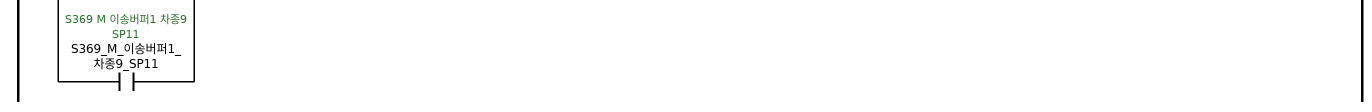
(* [picture p288: S369_유틸리티 rungs L95-L95] *)
(* S369_이송버퍼01 차종 유 *)
(* Rung L95 *)
IF (S369_M_이송버퍼1_차종1_AX OR S369_M_이송버퍼1_차종1_B OR S369_M_이송버퍼1_차종1_C OR S369_M_이송버퍼1_차종1_D OR S369_M_이송버퍼1_차종1_E OR S369_M_이송버퍼1_차종1_F OR S369_M_이송버퍼1_차종1_G OR S369_M_이송버퍼1_차종1_H) AND (S369_M_이송버퍼1_차종2_3DR OR S369_M_이송버퍼1_차종2_4DR OR S369_M_이송버퍼1_차종2_5DR OR S369_M_이송버퍼1_차종2_WGN OR S369_M_이송버퍼1_차종2_SP1 OR S369_M_이송버퍼1_차종2_SP2) AND (S369_M_이송버퍼1_차종3_LHD OR S369_M_이송버퍼1_차종3_RHD) AND (S369_M_이송버퍼1_차종4_내수 OR S369_M_이송버퍼1_차종4_수출 OR S369_M_이송버퍼1_차종4_북미 OR S369_M_이송버퍼1_차종4_EEC OR S369_M_이송버퍼1_차종4_호주 OR S369_M_이송버퍼1_차종4_중동 OR S369_M_이송버퍼1_차종4_중국 OR S369_M_이송버퍼1_차종4_브라질 OR S369_M_이송버퍼1_차종4_SP1 OR S369_M_이송버퍼1_차종4_SP2 OR S369_M_이송버퍼1_차종4_러시아 OR S369_M_이송버퍼1_차종4_SP3 OR S369_M_이송버퍼1_차종4_SP4 OR S369_M_이송버퍼1_차종4_SP5 OR S369_M_이송버퍼1_차종4_SP6 OR S369_M_이송버퍼1_차종4_SP7) AND (S369_M_이송버퍼1_차종5_MT OR S369_M_이송버퍼1_차종5_AT OR S369_M_이송버퍼1_차종5_SP1) AND (S369_M_이송버퍼1_차종6_일반루프 OR S369_M_이송버퍼1_차종6_썬루프 OR S369_M_이송버퍼1_차종6_파노라마루프 OR S369_M_이송버퍼1_차종6_DSROOF OR S369_M_이송버퍼1_차종6_SP1) AND (S369_M_이송버퍼1_차종7_GSL OR S369_M_이송버퍼1_차종7_DSL OR S369_M_이송버퍼1_차종7_SP1 OR S369_M_이송버퍼1_차종7_SP2 OR S369_M_이송버퍼1_차종7_SP3 OR S369_M_이송버퍼1_차종7_SP4 OR S369_M_이송버퍼1_차종7_SP5 OR S369_M_이송버퍼1_차종7_SP6) AND (S369_M_이송버퍼1_차종8_2WD OR S369_M_이송버퍼1_차종8_4WD OR S369_M_이송버퍼1_차종8_SP1) AND (S369_M_이송버퍼1_차종9_MPI OR S369_M_이송버퍼1_차종9_T_GDI OR S369_M_이송버퍼1_차종9_SP1 OR S369_M_이송버퍼1_차종9_SP2 OR S369_M_이송버퍼1_차종9_SP3 OR S369_M_이송버퍼1_차종9_SP4 OR S369_M_이송버퍼1_차종9_SP5 OR S369_M_이송버퍼1_차종9_SP6 OR S369_M_이송버퍼1_차종9_SP7 OR S369_M_이송버퍼1_차종9_SP8 OR S369_M_이송버퍼1_차종9_SP9 OR S369_M_이송버퍼1_차종9_SP10 OR S369_M_이송버퍼1_차종9_SP11) AND (S369_M_이송버퍼1_차종_OPT1_슬라이딩_유 OR S369_M_이송버퍼1_차종_OPT1_슬라이딩_무 OR S369_M_이송버퍼1_차종_OPT1_R_RACK_유 OR S369_M_이송버퍼1_차종_OPT1_R_RACK_무 OR S369_M_이송버퍼1_차종_OPT1_폴딩_유 OR S369_M_이송버퍼1_차종_OPT1_폴딩_무 OR S369_M_이송버퍼1_차종_OPT1_S_REP_EATER_유 OR S369_M_이송버퍼1_차종_OPT1_S_REP_EATER_무 OR S369_M_이송버퍼1_차종_OPT1_VAN_유 OR S369_M_이송버퍼1_차종_OPT1_VAN_무) THEN
    _t5 := S369_M_이송버퍼1_SEQ <> 0;
END_IF;
S369_M_이송버퍼1_차종_유 := _t5;

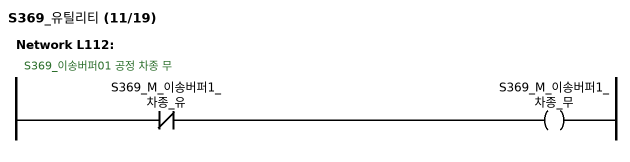
(* S369_이송버퍼01 공정 차종 무 *)
(* Rung L112 *)
S369_M_이송버퍼1_차종_무 := NOT S369_M_이송버퍼1_차종_유;

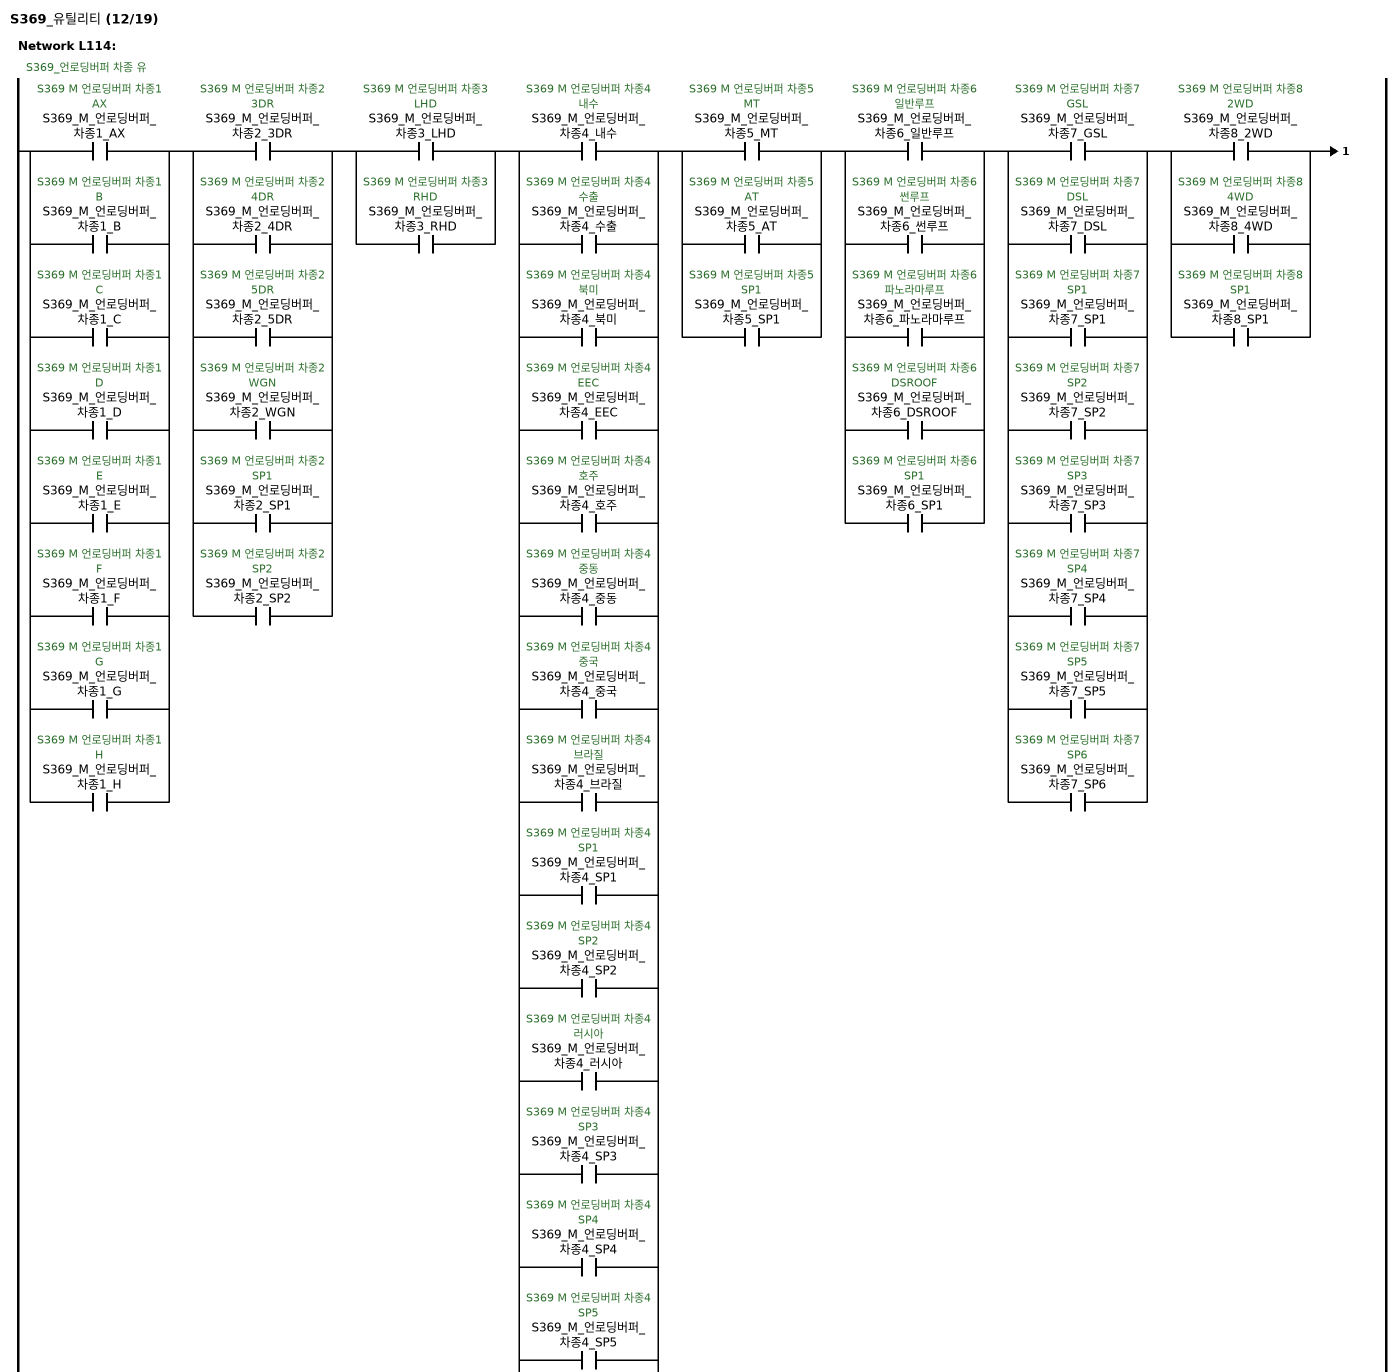

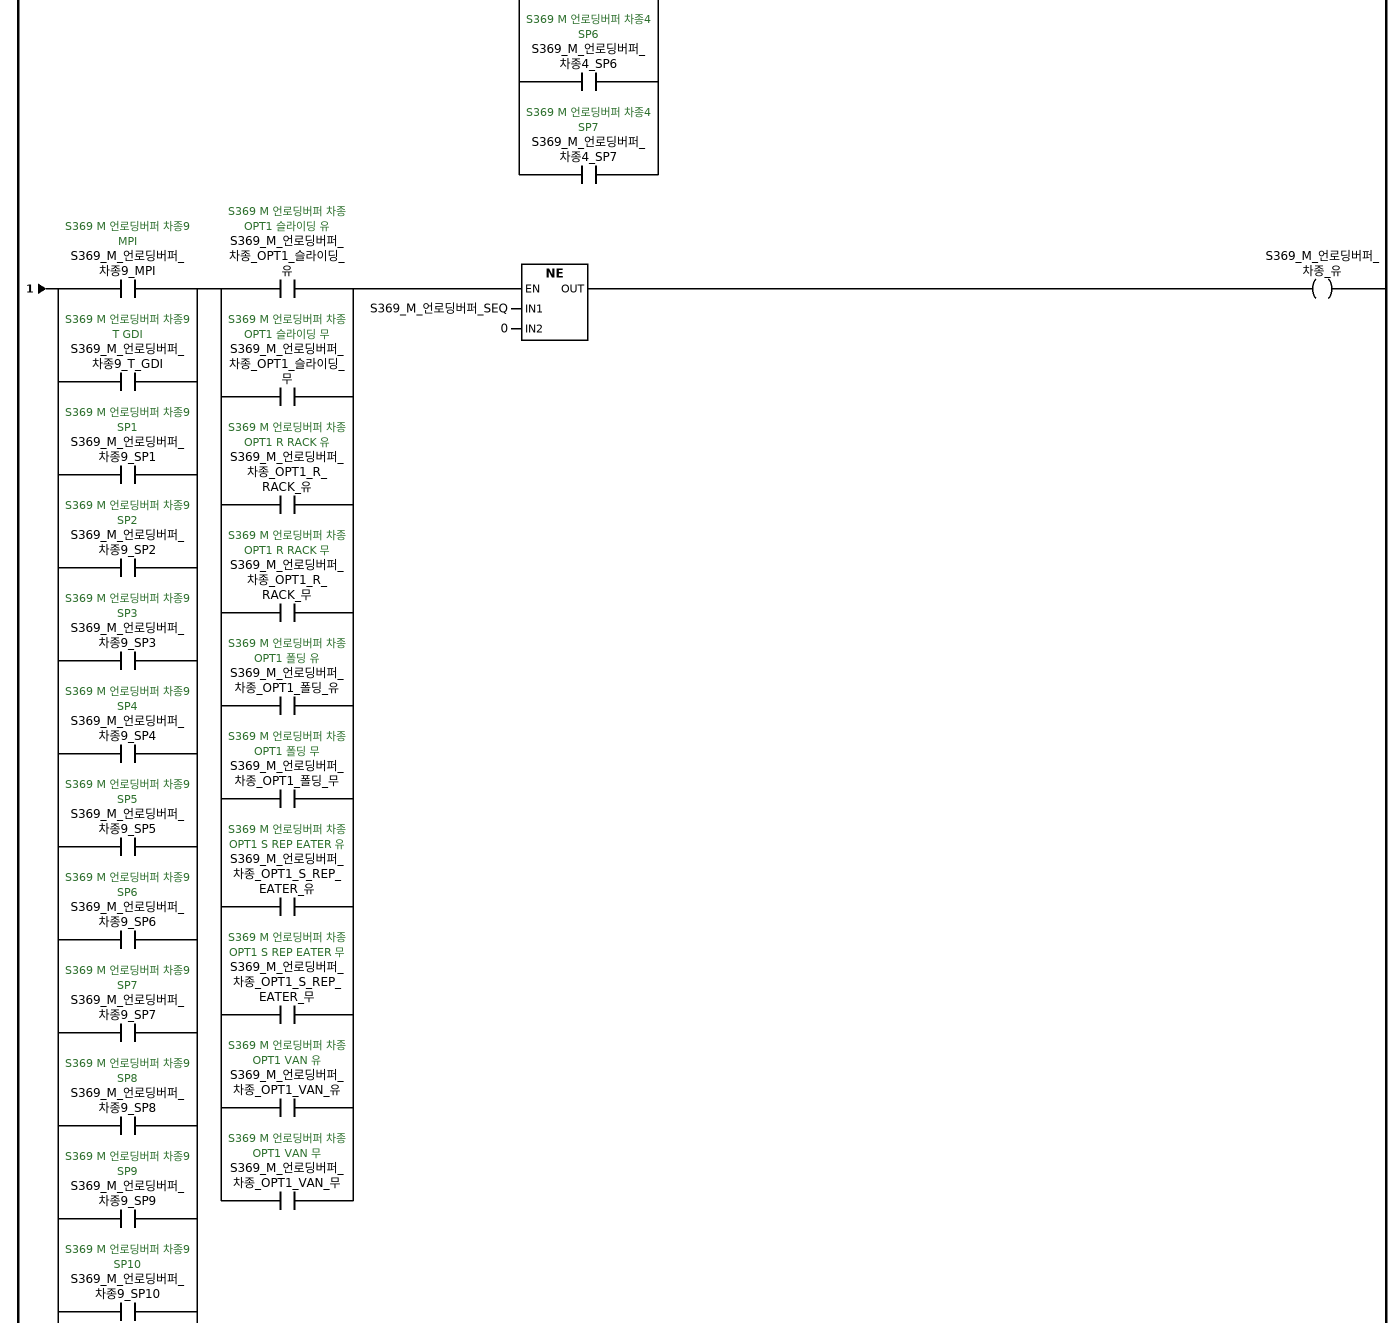

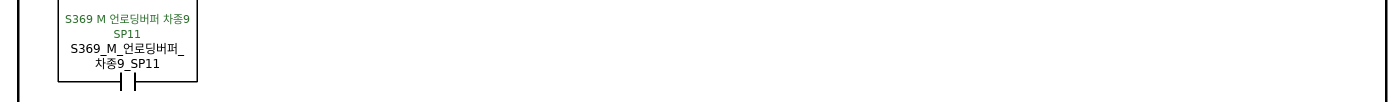
(* S369_언로딩버퍼 차종 유 *)
(* Rung L114 *)
IF (S369_M_언로딩버퍼_차종1_AX OR S369_M_언로딩버퍼_차종1_B OR S369_M_언로딩버퍼_차종1_C OR S369_M_언로딩버퍼_차종1_D OR S369_M_언로딩버퍼_차종1_E OR S369_M_언로딩버퍼_차종1_F OR S369_M_언로딩버퍼_차종1_G OR S369_M_언로딩버퍼_차종1_H) AND (S369_M_언로딩버퍼_차종2_3DR OR S369_M_언로딩버퍼_차종2_4DR OR S369_M_언로딩버퍼_차종2_5DR OR S369_M_언로딩버퍼_차종2_WGN OR S369_M_언로딩버퍼_차종2_SP1 OR S369_M_언로딩버퍼_차종2_SP2) AND (S369_M_언로딩버퍼_차종3_LHD OR S369_M_언로딩버퍼_차종3_RHD) AND (S369_M_언로딩버퍼_차종4_내수 OR S369_M_언로딩버퍼_차종4_수출 OR S369_M_언로딩버퍼_차종4_북미 OR S369_M_언로딩버퍼_차종4_EEC OR S369_M_언로딩버퍼_차종4_호주 OR S369_M_언로딩버퍼_차종4_중동 OR S369_M_언로딩버퍼_차종4_중국 OR S369_M_언로딩버퍼_차종4_브라질 OR S369_M_언로딩버퍼_차종4_SP1 OR S369_M_언로딩버퍼_차종4_SP2 OR S369_M_언로딩버퍼_차종4_러시아 OR S369_M_언로딩버퍼_차종4_SP3 OR S369_M_언로딩버퍼_차종4_SP4 OR S369_M_언로딩버퍼_차종4_SP5 OR S369_M_언로딩버퍼_차종4_SP6 OR S369_M_언로딩버퍼_차종4_SP7) AND (S369_M_언로딩버퍼_차종5_MT OR S369_M_언로딩버퍼_차종5_AT OR S369_M_언로딩버퍼_차종5_SP1) AND (S369_M_언로딩버퍼_차종6_일반루프 OR S369_M_언로딩버퍼_차종6_썬루프 OR S369_M_언로딩버퍼_차종6_파노라마루프 OR S369_M_언로딩버퍼_차종6_DSROOF OR S369_M_언로딩버퍼_차종6_SP1) AND (S369_M_언로딩버퍼_차종7_GSL OR S369_M_언로딩버퍼_차종7_DSL OR S369_M_언로딩버퍼_차종7_SP1 OR S369_M_언로딩버퍼_차종7_SP2 OR S369_M_언로딩버퍼_차종7_SP3 OR S369_M_언로딩버퍼_차종7_SP4 OR S369_M_언로딩버퍼_차종7_SP5 OR S369_M_언로딩버퍼_차종7_SP6) AND (S369_M_언로딩버퍼_차종8_2WD OR S369_M_언로딩버퍼_차종8_4WD OR S369_M_언로딩버퍼_차종8_SP1) AND (S369_M_언로딩버퍼_차종9_MPI OR S369_M_언로딩버퍼_차종9_T_GDI OR S369_M_언로딩버퍼_차종9_SP1 OR S369_M_언로딩버퍼_차종9_SP2 OR S369_M_언로딩버퍼_차종9_SP3 OR S369_M_언로딩버퍼_차종9_SP4 OR S369_M_언로딩버퍼_차종9_SP5 OR S369_M_언로딩버퍼_차종9_SP6 OR S369_M_언로딩버퍼_차종9_SP7 OR S369_M_언로딩버퍼_차종9_SP8 OR S369_M_언로딩버퍼_차종9_SP9 OR S369_M_언로딩버퍼_차종9_SP10 OR S369_M_언로딩버퍼_차종9_SP11) AND (S369_M_언로딩버퍼_차종_OPT1_슬라이딩_유 OR S369_M_언로딩버퍼_차종_OPT1_슬라이딩_무 OR S369_M_언로딩버퍼_차종_OPT1_R_RACK_유 OR S369_M_언로딩버퍼_차종_OPT1_R_RACK_무 OR S369_M_언로딩버퍼_차종_OPT1_폴딩_유 OR S369_M_언로딩버퍼_차종_OPT1_폴딩_무 OR S369_M_언로딩버퍼_차종_OPT1_S_REP_EATER_유 OR S369_M_언로딩버퍼_차종_OPT1_S_REP_EATER_무 OR S369_M_언로딩버퍼_차종_OPT1_VAN_유 OR S369_M_언로딩버퍼_차종_OPT1_VAN_무) THEN
    _t6 := S369_M_언로딩버퍼_SEQ <> 0;
END_IF;
S369_M_언로딩버퍼_차종_유 := _t6;

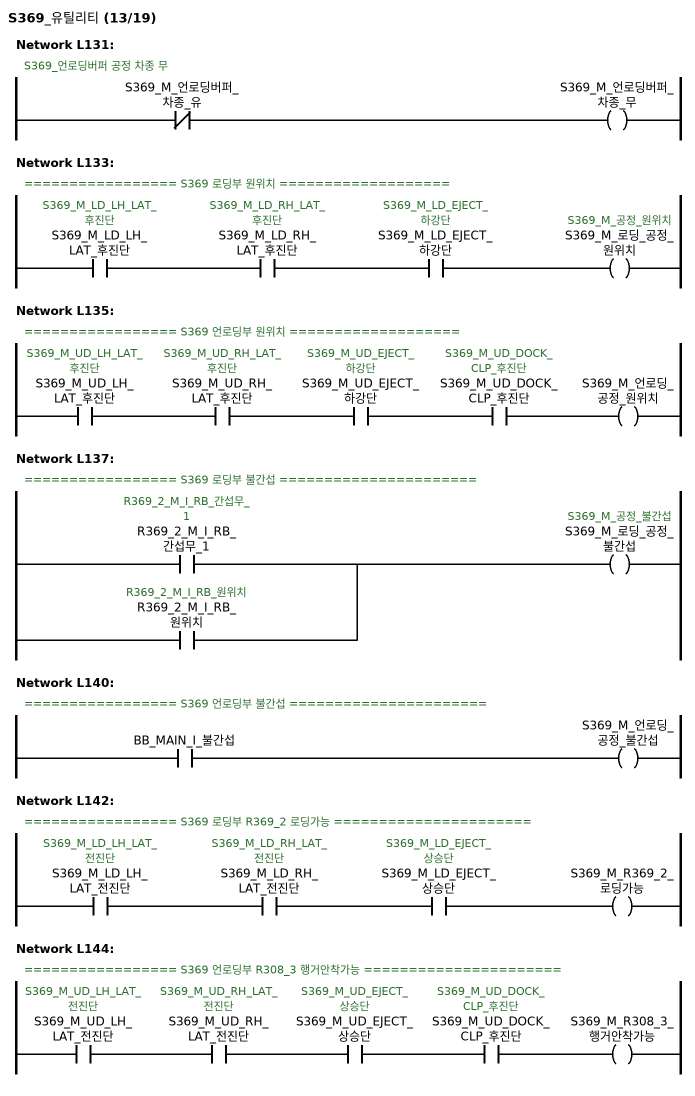
(* S369_언로딩버퍼 공정 차종 무 *)
(* Rung L131 *)
S369_M_언로딩버퍼_차종_무 := NOT S369_M_언로딩버퍼_차종_유;
(* ================= S369 로딩부 원위치 =================== *)
(* Rung L133 *)
S369_M_로딩_공정_원위치 := S369_M_LD_LH_LAT_후진단 AND S369_M_LD_RH_LAT_후진단 AND S369_M_LD_EJECT_하강단;
(* ================= S369 언로딩부 원위치 =================== *)
(* Rung L135 *)
S369_M_언로딩_공정_원위치 := S369_M_UD_LH_LAT_후진단 AND S369_M_UD_RH_LAT_후진단 AND S369_M_UD_EJECT_하강단 AND S369_M_UD_DOCK_CLP_후진단;
(* ================= S369 로딩부 불간섭 ====================== *)
(* Rung L137 *)
S369_M_로딩_공정_불간섭 := R369_2_M_I_RB_간섭무_1 OR R369_2_M_I_RB_원위치;
(* ================= S369 언로딩부 불간섭 ====================== *)
(* Rung L140 *)
S369_M_언로딩_공정_불간섭 := BB_MAIN_I_불간섭;
(* ================= S369 로딩부 R369_2 로딩가능 ====================== *)
(* Rung L142 *)
S369_M_R369_2_로딩가능 := S369_M_LD_LH_LAT_전진단 AND S369_M_LD_RH_LAT_전진단 AND S369_M_LD_EJECT_상승단;
(* ================= S369 언로딩부 R308_3 행거안착가능 ====================== *)
(* Rung L144 *)
S369_M_R308_3_행거안착가능 := S369_M_UD_LH_LAT_전진단 AND S369_M_UD_RH_LAT_전진단 AND S369_M_UD_EJECT_상승단 AND S369_M_UD_DOCK_CLP_후진단;

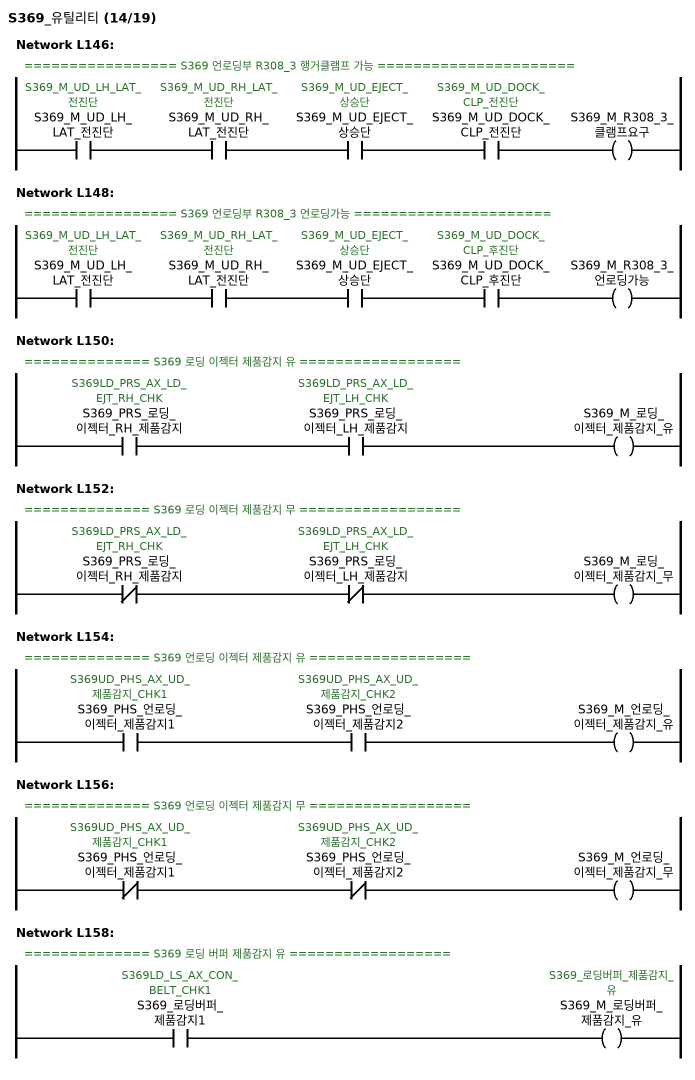
(* ================= S369 언로딩부 R308_3 행거클램프 가능 ====================== *)
(* Rung L146 *)
S369_M_R308_3_클램프요구 := S369_M_UD_LH_LAT_전진단 AND S369_M_UD_RH_LAT_전진단 AND S369_M_UD_EJECT_상승단 AND S369_M_UD_DOCK_CLP_전진단;
(* ================= S369 언로딩부 R308_3 언로딩가능 ====================== *)
(* Rung L148 *)
S369_M_R308_3_언로딩가능 := S369_M_UD_LH_LAT_전진단 AND S369_M_UD_RH_LAT_전진단 AND S369_M_UD_EJECT_상승단 AND S369_M_UD_DOCK_CLP_후진단;
(* ============== S369 로딩 이젝터 제품감지 유 ================== *)
(* Rung L150 *)
S369_M_로딩_이젝터_제품감지_유 := S369_PRS_로딩_이젝터_RH_제품감지 AND S369_PRS_로딩_이젝터_LH_제품감지;
(* ============== S369 로딩 이젝터 제품감지 무 ================== *)
(* Rung L152 *)
S369_M_로딩_이젝터_제품감지_무 := NOT S369_PRS_로딩_이젝터_RH_제품감지 AND NOT S369_PRS_로딩_이젝터_LH_제품감지;
(* ============== S369 언로딩 이젝터 제품감지 유 ================== *)
(* Rung L154 *)
S369_M_언로딩_이젝터_제품감지_유 := S369_PHS_언로딩_이젝터_제품감지1 AND S369_PHS_언로딩_이젝터_제품감지2;
(* ============== S369 언로딩 이젝터 제품감지 무 ================== *)
(* Rung L156 *)
S369_M_언로딩_이젝터_제품감지_무 := NOT S369_PHS_언로딩_이젝터_제품감지1 AND NOT S369_PHS_언로딩_이젝터_제품감지2;
(* ============== S369 로딩 버퍼 제품감지 유 ================== *)
(* Rung L158 *)
S369_M_로딩버퍼_제품감지_유 := S369_로딩버퍼_제품감지1;

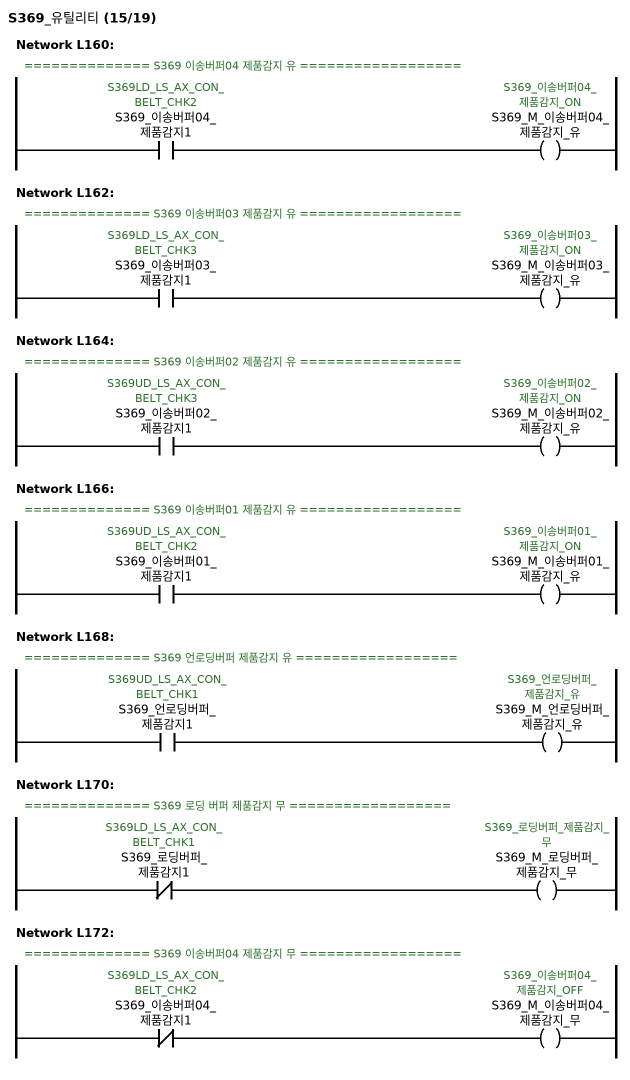
(* ============== S369 이송버퍼04 제품감지 유 ================== *)
(* Rung L160 *)
S369_M_이송버퍼04_제품감지_유 := S369_이송버퍼04_제품감지1;
(* ============== S369 이송버퍼03 제품감지 유 ================== *)
(* Rung L162 *)
S369_M_이송버퍼03_제품감지_유 := S369_이송버퍼03_제품감지1;
(* ============== S369 이송버퍼02 제품감지 유 ================== *)
(* Rung L164 *)
S369_M_이송버퍼02_제품감지_유 := S369_이송버퍼02_제품감지1;
(* ============== S369 이송버퍼01 제품감지 유 ================== *)
(* Rung L166 *)
S369_M_이송버퍼01_제품감지_유 := S369_이송버퍼01_제품감지1;
(* ============== S369 언로딩버퍼 제품감지 유 ================== *)
(* Rung L168 *)
S369_M_언로딩버퍼_제품감지_유 := S369_언로딩버퍼_제품감지1;
(* ============== S369 로딩 버퍼 제품감지 무 ================== *)
(* Rung L170 *)
S369_M_로딩버퍼_제품감지_무 := NOT S369_로딩버퍼_제품감지1;
(* ============== S369 이송버퍼04 제품감지 무 ================== *)
(* Rung L172 *)
S369_M_이송버퍼04_제품감지_무 := NOT S369_이송버퍼04_제품감지1;

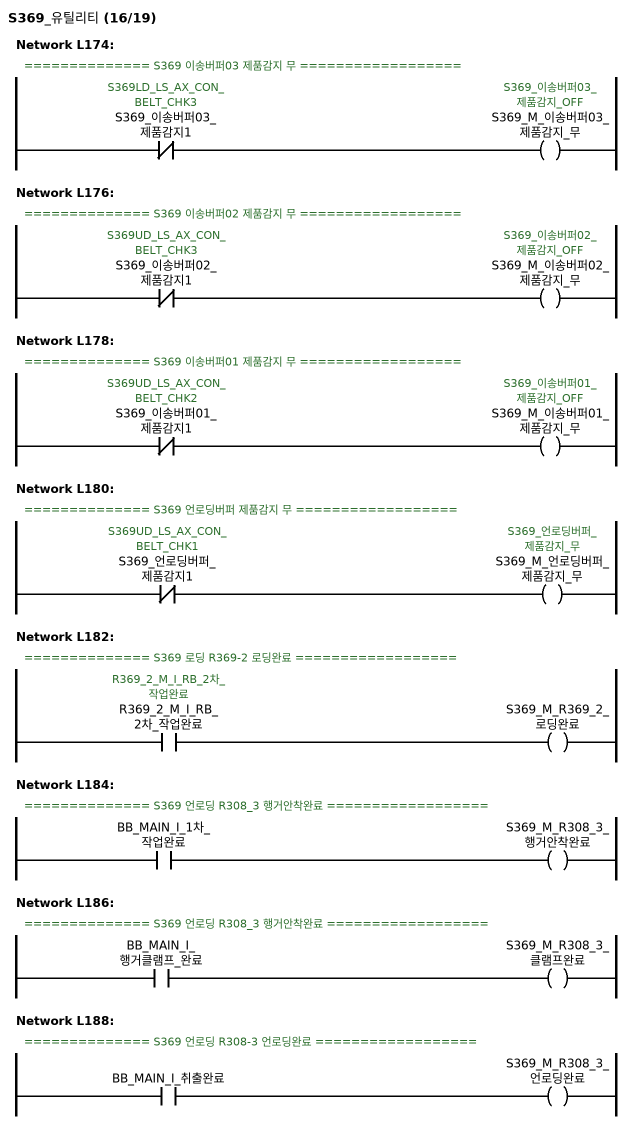
(* ============== S369 이송버퍼03 제품감지 무 ================== *)
(* Rung L174 *)
S369_M_이송버퍼03_제품감지_무 := NOT S369_이송버퍼03_제품감지1;
(* ============== S369 이송버퍼02 제품감지 무 ================== *)
(* Rung L176 *)
S369_M_이송버퍼02_제품감지_무 := NOT S369_이송버퍼02_제품감지1;
(* ============== S369 이송버퍼01 제품감지 무 ================== *)
(* Rung L178 *)
S369_M_이송버퍼01_제품감지_무 := NOT S369_이송버퍼01_제품감지1;
(* ============== S369 언로딩버퍼 제품감지 무 ================== *)
(* Rung L180 *)
S369_M_언로딩버퍼_제품감지_무 := NOT S369_언로딩버퍼_제품감지1;
(* ============== S369 로딩 R369-2 로딩완료 ================== *)
(* Rung L182 *)
S369_M_R369_2_로딩완료 := R369_2_M_I_RB_2차_작업완료;
(* ============== S369 언로딩 R308_3 행거안착완료 ================== *)
(* Rung L184 *)
S369_M_R308_3_행거안착완료 := BB_MAIN_I_1차_작업완료;
(* ============== S369 언로딩 R308_3 행거안착완료 ================== *)
(* Rung L186 *)
S369_M_R308_3_클램프완료 := BB_MAIN_I_행거클램프_완료;
(* ============== S369 언로딩 R308-3 언로딩완료 ================== *)
(* Rung L188 *)
S369_M_R308_3_언로딩완료 := BB_MAIN_I_취출완료;

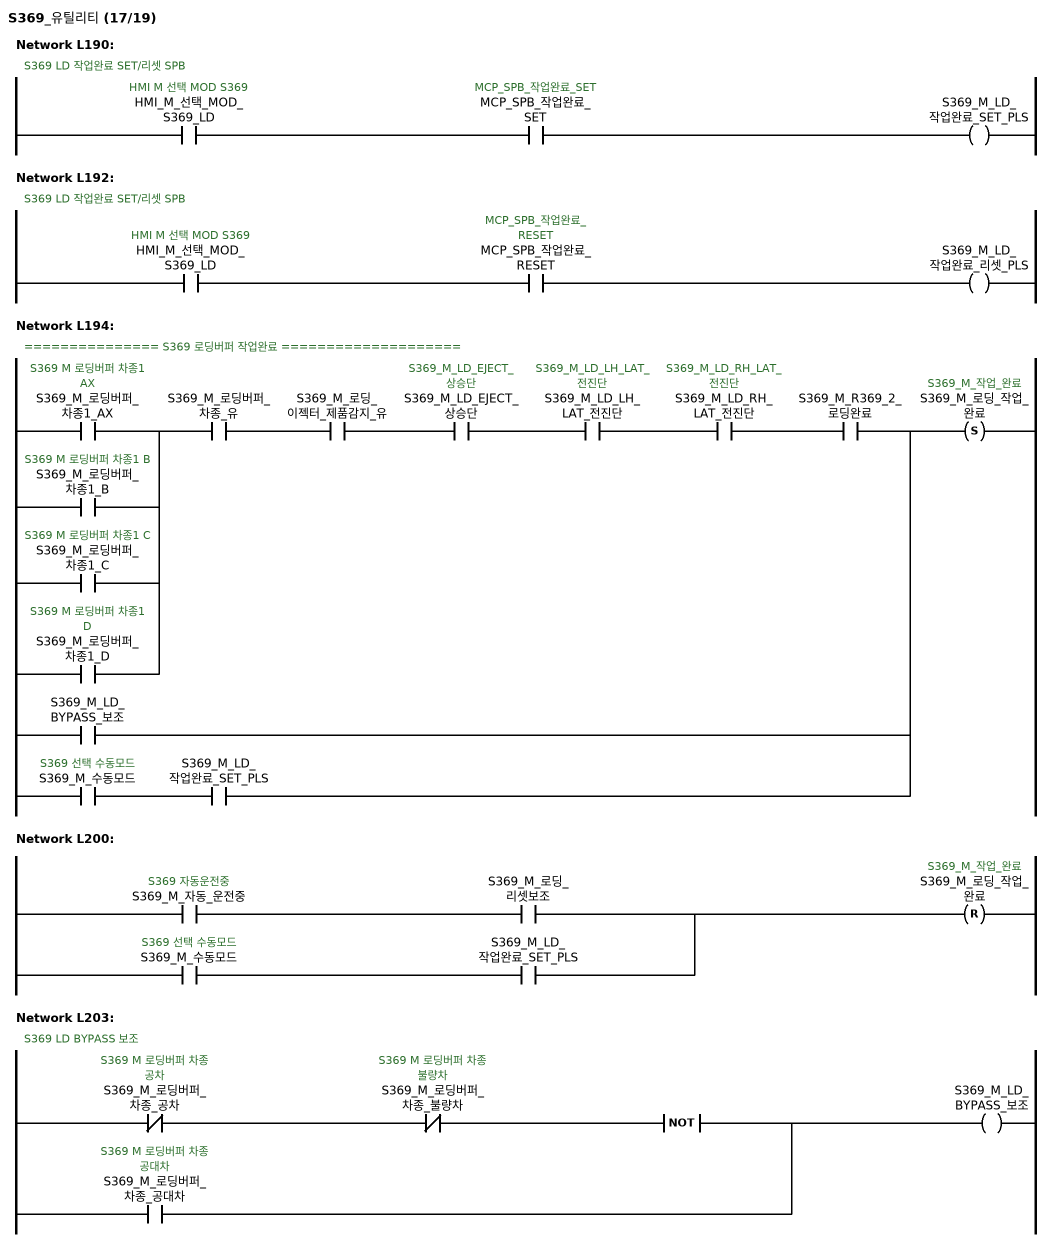
(* S369 LD 작업완료 SET/리셋 SPB *)
(* Rung L190 *)
S369_M_LD_작업완료_SET_PLS := HMI_M_선택_MOD_S369_LD AND MCP_SPB_작업완료_SET;
(* S369 LD 작업완료 SET/리셋 SPB *)
(* Rung L192 *)
S369_M_LD_작업완료_리셋_PLS := HMI_M_선택_MOD_S369_LD AND MCP_SPB_작업완료_RESET;
(* =============== S369 로딩버퍼 작업완료 ==================== *)
(* Rung L194 *)
IF ((S369_M_로딩버퍼_차종1_AX OR S369_M_로딩버퍼_차종1_B OR S369_M_로딩버퍼_차종1_C OR S369_M_로딩버퍼_차종1_D) AND S369_M_로딩버퍼_차종_유 AND S369_M_로딩_이젝터_제품감지_유 AND S369_M_LD_EJECT_상승단 AND S369_M_LD_LH_LAT_전진단 AND S369_M_LD_RH_LAT_전진단 AND S369_M_R369_2_로딩완료) OR S369_M_LD_BYPASS_보조 OR (S369_M_수동모드 AND S369_M_LD_작업완료_SET_PLS) THEN
    S369_M_로딩_작업_완료 := TRUE;
END_IF;
(* Rung L200 *)
IF (S369_M_자동_운전중 AND S369_M_로딩_리셋보조) OR (S369_M_수동모드 AND S369_M_LD_작업완료_SET_PLS) THEN
    S369_M_로딩_작업_완료 := FALSE;
END_IF;
(* S369 LD BYPASS 보조 *)
(* Rung L203 *)
S369_M_LD_BYPASS_보조 := NOT (NOT S369_M_로딩버퍼_차종_공차 AND NOT S369_M_로딩버퍼_차종_불량차) OR S369_M_로딩버퍼_차종_공대차;

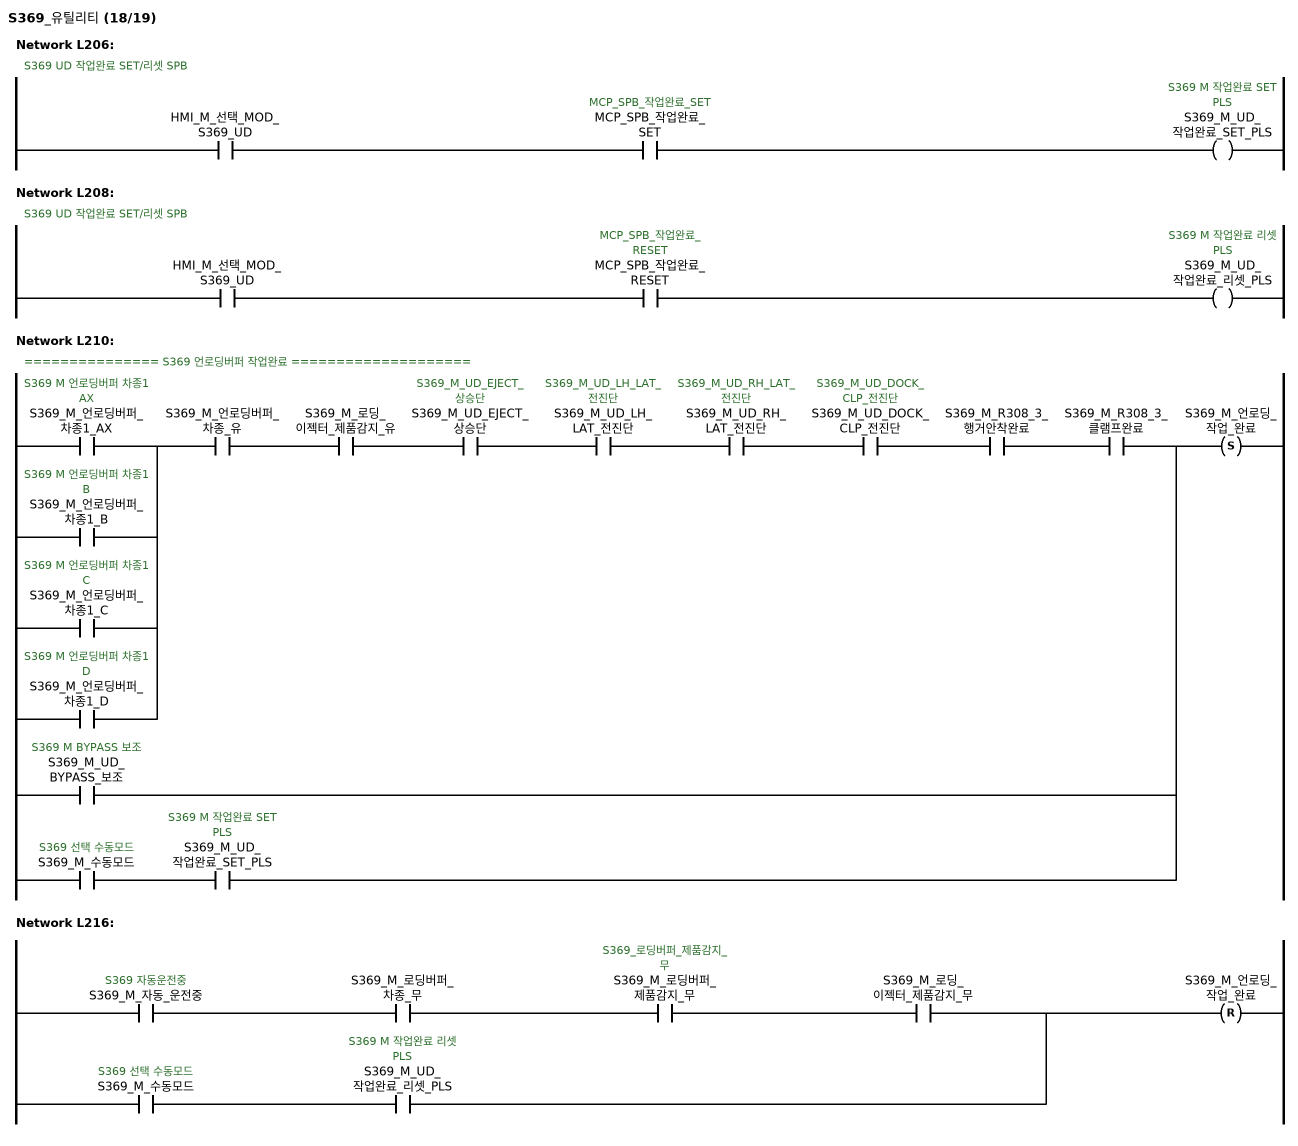
(* S369 UD 작업완료 SET/리셋 SPB *)
(* Rung L206 *)
S369_M_UD_작업완료_SET_PLS := HMI_M_선택_MOD_S369_UD AND MCP_SPB_작업완료_SET;
(* S369 UD 작업완료 SET/리셋 SPB *)
(* Rung L208 *)
S369_M_UD_작업완료_리셋_PLS := HMI_M_선택_MOD_S369_UD AND MCP_SPB_작업완료_RESET;
(* =============== S369 언로딩버퍼 작업완료 ==================== *)
(* Rung L210 *)
IF ((S369_M_언로딩버퍼_차종1_AX OR S369_M_언로딩버퍼_차종1_B OR S369_M_언로딩버퍼_차종1_C OR S369_M_언로딩버퍼_차종1_D) AND S369_M_언로딩버퍼_차종_유 AND S369_M_로딩_이젝터_제품감지_유 AND S369_M_UD_EJECT_상승단 AND S369_M_UD_LH_LAT_전진단 AND S369_M_UD_RH_LAT_전진단 AND S369_M_UD_DOCK_CLP_전진단 AND S369_M_R308_3_행거안착완료 AND S369_M_R308_3_클램프완료) OR S369_M_UD_BYPASS_보조 OR (S369_M_수동모드 AND S369_M_UD_작업완료_SET_PLS) THEN
    S369_M_언로딩_작업_완료 := TRUE;
END_IF;
(* Rung L216 *)
IF (S369_M_자동_운전중 AND S369_M_로딩버퍼_차종_무 AND S369_M_로딩버퍼_제품감지_무 AND S369_M_로딩_이젝터_제품감지_무) OR (S369_M_수동모드 AND S369_M_UD_작업완료_리셋_PLS) THEN
    S369_M_언로딩_작업_완료 := FALSE;
END_IF;

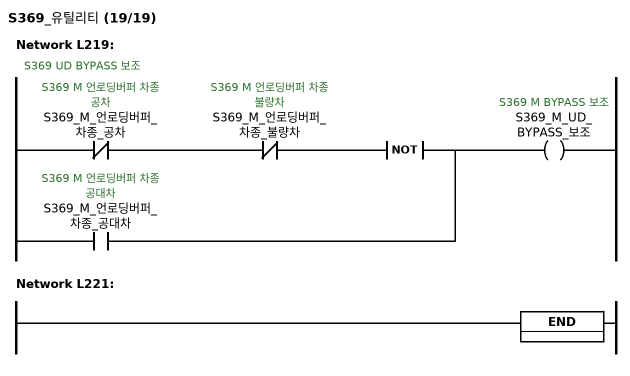
(* S369 UD BYPASS 보조 *)
(* Rung L219 *)
S369_M_UD_BYPASS_보조 := NOT (NOT S369_M_언로딩버퍼_차종_공차 AND NOT S369_M_언로딩버퍼_차종_불량차) OR S369_M_언로딩버퍼_차종_공대차;
(* Rung L221 *)
END();
END_PROGRAM

PROGRAM S369_동작 (* task: 스캔 프로그램 *)
VAR_EXTERNAL RETAIN
    ALWAYS_ON : BOOL; (* AT %MW3.1 *) (* 항시 ON *)
    S369_HOME : BOOL; (* AT %MW5048.0 *) (* S369_HOME *)
    S369_M_LD_EJECT_상승_LS_이상 : BOOL; (* AT %MW5100.5 *) (* S369_M_LD_EJECT_상승_LS_이상 *)
    S369_M_LD_EJECT_상승_보조 : BOOL; (* AT %MW5100.1 *) (* S369_M_LD_EJECT_상승_보조 *)
    S369_M_LD_EJECT_상승단 : BOOL; (* AT %MW5100.3 *) (* S369_M_LD_EJECT_상승단 *)
    S369_M_LD_EJECT_조건 : BOOL; (* AT %MW5100.0 *) (* S369_M_LD_EJECT_조건 *)
    S369_M_LD_EJECT_하강_LS_이상 : BOOL; (* AT %MW5100.6 *) (* S369_M_LD_EJECT_하강_LS_이상 *)
    S369_M_LD_EJECT_하강_보조 : BOOL; (* AT %MW5100.2 *) (* S369_M_LD_EJECT_하강_보조 *)
    S369_M_LD_EJECT_하강단 : BOOL; (* AT %MW5100.4 *) (* S369_M_LD_EJECT_하강단 *)
    S369_M_LD_LH_LAT_전진_LS_이상 : BOOL; (* AT %MW5101.5 *) (* S369_M_LD_LH_LAT_전진_LS_이상 *)
    S369_M_LD_LH_LAT_전진_보조 : BOOL; (* AT %MW5101.1 *) (* S369_M_LD_LH_LAT_전진_보조 *)
    S369_M_LD_LH_LAT_전진단 : BOOL; (* AT %MW5101.3 *) (* S369_M_LD_LH_LAT_전진단 *)
    S369_M_LD_LH_LAT_조건 : BOOL; (* AT %MW5101.0 *) (* S369_M_LD_LH_LAT_조건 *)
    S369_M_LD_LH_LAT_후진_LS_이상 : BOOL; (* AT %MW5101.6 *) (* S369_M_LD_LH_LAT_후진_LS_이상 *)
    S369_M_LD_LH_LAT_후진_보조 : BOOL; (* AT %MW5101.2 *) (* S369_M_LD_LH_LAT_후진_보조 *)
    S369_M_LD_LH_LAT_후진단 : BOOL; (* AT %MW5101.4 *) (* S369_M_LD_LH_LAT_후진단 *)
    S369_M_LD_RH_LAT_전진_LS_이상 : BOOL; (* AT %MW5102.5 *) (* S369_M_LD_RH_LAT_전진_LS_이상 *)
    S369_M_LD_RH_LAT_전진_보조 : BOOL; (* AT %MW5102.1 *) (* S369_M_LD_RH_LAT_전진_보조 *)
    S369_M_LD_RH_LAT_전진단 : BOOL; (* AT %MW5102.3 *) (* S369_M_LD_RH_LAT_전진단 *)
    S369_M_LD_RH_LAT_조건 : BOOL; (* AT %MW5102.0 *) (* S369_M_LD_RH_LAT_조건 *)
    S369_M_LD_RH_LAT_후진_LS_이상 : BOOL; (* AT %MW5102.6 *) (* S369_M_LD_RH_LAT_후진_LS_이상 *)
    S369_M_LD_RH_LAT_후진_보조 : BOOL; (* AT %MW5102.2 *) (* S369_M_LD_RH_LAT_후진_보조 *)
    S369_M_LD_RH_LAT_후진단 : BOOL; (* AT %MW5102.4 *) (* S369_M_LD_RH_LAT_후진단 *)
    S369_M_R308_3_클램프완료 : BOOL; (* AT %MW5001.4 *)
    S369_M_R308_3_행거안착완료 : BOOL; (* AT %MW5001.3 *)
    S369_M_R369_2_로딩완료 : BOOL; (* AT %MW5001.2 *)
    S369_M_UD_DOCK_CLP_전진_LS_이상 : BOOL; (* AT %MW5111.5 *) (* S369_M_UD_DOCK_CLP_전진_LS_이상 *)
    S369_M_UD_DOCK_CLP_전진_보조 : BOOL; (* AT %MW5111.1 *) (* S369_M_UD_DOCK_CLP_전진_보조 *)
    S369_M_UD_DOCK_CLP_전진단 : BOOL; (* AT %MW5111.3 *) (* S369_M_UD_DOCK_CLP_전진단 *)
    S369_M_UD_DOCK_CLP_조건 : BOOL; (* AT %MW5111.0 *) (* S369_M_UD_DOCK_CLP_조건 *)
    S369_M_UD_DOCK_CLP_후진_LS_이상 : BOOL; (* AT %MW5111.6 *) (* S369_M_UD_DOCK_CLP_후진_LS_이상 *)
    S369_M_UD_DOCK_CLP_후진_보조 : BOOL; (* AT %MW5111.2 *) (* S369_M_UD_DOCK_CLP_후진_보조 *)
    S369_M_UD_DOCK_CLP_후진단 : BOOL; (* AT %MW5111.4 *) (* S369_M_UD_DOCK_CLP_후진단 *)
    S369_M_UD_EJECT_상승_LS_이상 : BOOL; (* AT %MW5108.5 *) (* S369_M_UD_EJECT_상승_LS_이상 *)
    S369_M_UD_EJECT_상승_보조 : BOOL; (* AT %MW5108.1 *) (* S369_M_UD_EJECT_상승_보조 *)
    S369_M_UD_EJECT_상승단 : BOOL; (* AT %MW5108.3 *) (* S369_M_UD_EJECT_상승단 *)
    S369_M_UD_EJECT_조건 : BOOL; (* AT %MW5108.0 *) (* S369_M_UD_EJECT_조건 *)
    S369_M_UD_EJECT_하강_LS_이상 : BOOL; (* AT %MW5108.6 *) (* S369_M_UD_EJECT_하강_LS_이상 *)
    S369_M_UD_EJECT_하강_보조 : BOOL; (* AT %MW5108.2 *) (* S369_M_UD_EJECT_하강_보조 *)
    S369_M_UD_EJECT_하강단 : BOOL; (* AT %MW5108.4 *) (* S369_M_UD_EJECT_하강단 *)
    S369_M_UD_LH_LAT_전진_LS_이상 : BOOL; (* AT %MW5109.5 *) (* S369_M_UD_LH_LAT_전진_LS_이상 *)
    S369_M_UD_LH_LAT_전진_보조 : BOOL; (* AT %MW5109.1 *) (* S369_M_UD_LH_LAT_전진_보조 *)
    S369_M_UD_LH_LAT_전진단 : BOOL; (* AT %MW5109.3 *) (* S369_M_UD_LH_LAT_전진단 *)
    S369_M_UD_LH_LAT_조건 : BOOL; (* AT %MW5109.0 *) (* S369_M_UD_LH_LAT_조건 *)
    S369_M_UD_LH_LAT_후진_LS_이상 : BOOL; (* AT %MW5109.6 *) (* S369_M_UD_LH_LAT_후진_LS_이상 *)
    S369_M_UD_LH_LAT_후진_보조 : BOOL; (* AT %MW5109.2 *) (* S369_M_UD_LH_LAT_후진_보조 *)
    S369_M_UD_LH_LAT_후진단 : BOOL; (* AT %MW5109.4 *) (* S369_M_UD_LH_LAT_후진단 *)
    S369_M_UD_RH_LAT_전진_LS_이상 : BOOL; (* AT %MW5110.5 *) (* S369_M_UD_RH_LAT_전진_LS_이상 *)
    S369_M_UD_RH_LAT_전진_보조 : BOOL; (* AT %MW5110.1 *) (* S369_M_UD_RH_LAT_전진_보조 *)
    S369_M_UD_RH_LAT_전진단 : BOOL; (* AT %MW5110.3 *) (* S369_M_UD_RH_LAT_전진단 *)
    S369_M_UD_RH_LAT_조건 : BOOL; (* AT %MW5110.0 *) (* S369_M_UD_RH_LAT_조건 *)
    S369_M_UD_RH_LAT_후진_LS_이상 : BOOL; (* AT %MW5110.6 *) (* S369_M_UD_RH_LAT_후진_LS_이상 *)
    S369_M_UD_RH_LAT_후진_보조 : BOOL; (* AT %MW5110.2 *) (* S369_M_UD_RH_LAT_후진_보조 *)
    S369_M_UD_RH_LAT_후진단 : BOOL; (* AT %MW5110.4 *) (* S369_M_UD_RH_LAT_후진단 *)
    S369_M_동작_선택_1 : BOOL; (* AT %MW5040.0 *) (* S369_M_동작_선택_1 *)
    S369_M_동작_선택_10 : BOOL; (* AT %MW5040.9 *) (* S369_M_동작_선택_10 *)
    S369_M_동작_선택_11 : BOOL; (* AT %MW5040.10 *) (* S369_M_동작_선택_11 *)
    S369_M_동작_선택_12 : BOOL; (* AT %MW5040.11 *) (* S369_M_동작_선택_12 *)
    S369_M_동작_선택_2 : BOOL; (* AT %MW5040.1 *) (* S369_M_동작_선택_2 *)
    S369_M_동작_선택_3 : BOOL; (* AT %MW5040.2 *) (* S369_M_동작_선택_3 *)
    S369_M_동작_선택_9 : BOOL; (* AT %MW5040.8 *) (* S369_M_동작_선택_9 *)
    S369_M_로딩_공정_불간섭 : BOOL; (* AT %MW5004.2 *) (* S369_M_공정_불간섭 *)
    S369_M_로딩_이젝터_제품감지_무 : BOOL; (* AT %MW5001.9 *)
    S369_M_로딩_이젝터_제품감지_유 : BOOL; (* AT %MW5001.8 *)
    S369_M_로딩_작업_완료 : BOOL; (* AT %MW5001.0 *) (* S369_M_작업_완료 *)
    S369_M_로딩버퍼_제품감지_무 : BOOL; (* AT %MW5005.1 *) (* S369_로딩버퍼_제품감지_무 *)
    S369_M_로딩버퍼_차종_무 : BOOL; (* AT %MW5002.1 *)
    S369_M_로딩버퍼_차종_유 : BOOL; (* AT %MW5002.0 *)
    S369_M_수동모드 : BOOL; (* AT %MW5000.3 *) (* S369 선택 수동모드 *)
    S369_M_언로딩_공정_불간섭 : BOOL; (* AT %MW5004.3 *)
    S369_M_언로딩_이젝터_제품감지_무 : BOOL; (* AT %MW5001.11 *)
    S369_M_언로딩_이젝터_제품감지_유 : BOOL; (* AT %MW5001.10 *)
    S369_M_언로딩_작업_완료 : BOOL; (* AT %MW5001.1 *)
    S369_M_언로딩버퍼_도착완료 : BOOL; (* AT %MW5003.6 *)
    S369_M_언로딩버퍼_제품감지_무 : BOOL; (* AT %MW5005.11 *) (* S369_언로딩버퍼_제품감지_무 *)
    S369_M_언로딩버퍼_제품감지_유 : BOOL; (* AT %MW5005.10 *) (* S369_언로딩버퍼_제품감지_유 *)
    S369_M_언로딩버퍼_차종_무 : BOOL; (* AT %MW5002.3 *)
    S369_M_언로딩버퍼_차종_유 : BOOL; (* AT %MW5002.2 *)
    S369_M_운전준비_ON : BOOL; (* AT %MW5000.0 *) (* S369 운전준비 ON *)
    S369_M_자동_운전중 : BOOL; (* AT %MW5000.4 *) (* S369 자동운전중 *)
    S369_전진_ON : BOOL; (* AT %MW5048.1 *) (* S369_전진_ON *)
    S369_후진_ON : BOOL; (* AT %MW5048.2 *) (* S369_후진_ON *)
    전체_M_이상_리셋 : BOOL; (* AT %MW308.2 *) (* ALL공정 PB 이상리셋 *)
END_VAR
VAR_EXTERNAL
    EGIS_CWS : BOOL;
    S369LD_RS_AX_LH_LATCH_전진 : BOOL; (* AT %MW86411.0 *) (* S369LD_RS_AX_LH_LATCH_전진 *)
    S369LD_RS_AX_LH_LATCH_후진1 : BOOL; (* AT %MW86411.1 *) (* S369LD_RS_AX_LH_LATCH_후진1 *)
    S369LD_RS_AX_LH_LATCH_후진2 : BOOL; (* AT %MW86411.2 *) (* S369LD_RS_AX_LH_LATCH_후진2 *)
    S369LD_RS_AX_LH_LATCH_후진3 : BOOL; (* AT %MW86411.3 *) (* S369LD_RS_AX_LH_LATCH_후진3 *)
    S369LD_RS_AX_LH_LATCH_후진4 : BOOL; (* AT %MW86411.4 *) (* S369LD_RS_AX_LH_LATCH_후진4 *)
    S369LD_RS_AX_RH_LATCH_전진 : BOOL; (* AT %MW86410.8 *) (* S369LD_RS_AX_RH_LATCH_전진 *)
    S369LD_RS_AX_RH_LATCH_후진1 : BOOL; (* AT %MW86410.9 *) (* S369LD_RS_AX_RH_LATCH_후진1 *)
    S369LD_RS_AX_RH_LATCH_후진2 : BOOL; (* AT %MW86410.10 *) (* S369LD_RS_AX_RH_LATCH_후진2 *)
    S369LD_RS_AX_RH_LATCH_후진3 : BOOL; (* AT %MW86410.11 *) (* S369LD_RS_AX_RH_LATCH_후진3 *)
    S369LD_RS_AX_RH_LATCH_후진4 : BOOL; (* AT %MW86410.12 *) (* S369LD_RS_AX_RH_LATCH_후진4 *)
    S369LD_RS_EJECT_상승1 : BOOL; (* AT %MW86410.0 *) (* S369LD_RS_EJECT_상승1 *)
    S369LD_RS_EJECT_상승2 : BOOL; (* AT %MW86410.2 *) (* S369LD_RS_EJECT_상승2 *)
    S369LD_RS_EJECT_하강1 : BOOL; (* AT %MW86410.1 *) (* S369LD_RS_EJECT_하강1 *)
    S369LD_RS_EJECT_하강2 : BOOL; (* AT %MW86410.3 *) (* S369LD_RS_EJECT_하강2 *)
    S369LD_SOL_AX_LH_LATCH_전진 : BOOL; (* AT %MW96413.4 *) (* S369LD_SOL_AX_LH_LATCH_전진 *)
    S369LD_SOL_AX_LH_LATCH_후진 : BOOL; (* AT %MW96413.5 *) (* S369LD_SOL_AX_LH_LATCH_후진 *)
    S369LD_SOL_AX_RH_LATCH_전진 : BOOL; (* AT %MW96413.2 *) (* S369LD_SOL_AX_RH_LATCH_전진 *)
    S369LD_SOL_AX_RH_LATCH_후진 : BOOL; (* AT %MW96413.3 *) (* S369LD_SOL_AX_RH_LATCH_후진 *)
    S369LD_SOL_EJECT_상승 : BOOL; (* AT %MW96413.0 *) (* S369LD_SOL_EJECT_상승 *)
    S369LD_SOL_EJECT_하강 : BOOL; (* AT %MW96413.1 *) (* S369LD_SOL_EJECT_하강 *)
    S369UD_RS_AX_DOCK_CLP_전진 : BOOL; (* AT %MW86421.8 *) (* S369UD_RS_AX_DOCK_CLP_전진 *)
    S369UD_RS_AX_DOCK_CLP_후진1 : BOOL; (* AT %MW86421.9 *) (* S369UD_RS_AX_DOCK_CLP_후진1 *)
    S369UD_RS_AX_DOCK_CLP_후진2 : BOOL; (* AT %MW86421.10 *) (* S369UD_RS_AX_DOCK_CLP_후진2 *)
    S369UD_RS_AX_DOCK_CLP_후진3 : BOOL; (* AT %MW86421.11 *) (* S369UD_RS_AX_DOCK_CLP_후진3 *)
    S369UD_RS_AX_DOCK_CLP_후진4 : BOOL; (* AT %MW86421.12 *) (* S369UD_RS_AX_DOCK_CLP_후진4 *)
    S369UD_RS_AX_LH_LATCH_전진 : BOOL; (* AT %MW86421.0 *) (* S369UD_RS_AX_LH_LATCH_전진 *)
    S369UD_RS_AX_LH_LATCH_후진1 : BOOL; (* AT %MW86421.1 *) (* S369UD_RS_AX_LH_LATCH_후진1 *)
    S369UD_RS_AX_LH_LATCH_후진2 : BOOL; (* AT %MW86421.2 *) (* S369UD_RS_AX_LH_LATCH_후진2 *)
    S369UD_RS_AX_LH_LATCH_후진3 : BOOL; (* AT %MW86421.3 *) (* S369UD_RS_AX_LH_LATCH_후진3 *)
    S369UD_RS_AX_LH_LATCH_후진4 : BOOL; (* AT %MW86421.4 *) (* S369UD_RS_AX_LH_LATCH_후진4 *)
    S369UD_RS_AX_RH_LATCH_전진 : BOOL; (* AT %MW86420.8 *) (* S369UD_RS_AX_RH_LATCH_전진 *)
    S369UD_RS_AX_RH_LATCH_후진1 : BOOL; (* AT %MW86420.9 *) (* S369UD_RS_AX_RH_LATCH_후진1 *)
    S369UD_RS_AX_RH_LATCH_후진2 : BOOL; (* AT %MW86420.10 *) (* S369UD_RS_AX_RH_LATCH_후진2 *)
    S369UD_RS_AX_RH_LATCH_후진3 : BOOL; (* AT %MW86420.11 *) (* S369UD_RS_AX_RH_LATCH_후진3 *)
    S369UD_RS_AX_RH_LATCH_후진4 : BOOL; (* AT %MW86420.12 *) (* S369UD_RS_AX_RH_LATCH_후진4 *)
    S369UD_RS_EJECT_상승1 : BOOL; (* AT %MW86420.0 *) (* S369UD_RS_EJECT_상승1 *)
    S369UD_RS_EJECT_상승2 : BOOL; (* AT %MW86420.2 *) (* S369UD_RS_EJECT_상승2 *)
    S369UD_RS_EJECT_하강1 : BOOL; (* AT %MW86420.1 *) (* S369UD_RS_EJECT_하강1 *)
    S369UD_RS_EJECT_하강2 : BOOL; (* AT %MW86420.3 *) (* S369UD_RS_EJECT_하강2 *)
    S369UD_SOL_AX_DOCK_CLP_전진 : BOOL; (* AT %MW96423.6 *) (* S369UD_SOL_AX_DOCK_CLP_전진 *)
    S369UD_SOL_AX_DOCK_CLP_후진 : BOOL; (* AT %MW96423.7 *) (* S369UD_SOL_AX_DOCK_CLP_후진 *)
    S369UD_SOL_AX_LH_LATCH_전진 : BOOL; (* AT %MW96423.4 *) (* S369UD_SOL_AX_LH_LATCH_전진 *)
    S369UD_SOL_AX_LH_LATCH_후진 : BOOL; (* AT %MW96423.5 *) (* S369UD_SOL_AX_LH_LATCH_후진 *)
    S369UD_SOL_AX_RH_LATCH_전진 : BOOL; (* AT %MW96423.2 *) (* S369UD_SOL_AX_RH_LATCH_전진 *)
    S369UD_SOL_AX_RH_LATCH_후진 : BOOL; (* AT %MW96423.3 *) (* S369UD_SOL_AX_RH_LATCH_후진 *)
    S369UD_SOL_EJECT_상승 : BOOL; (* AT %MW96423.0 *) (* S369UD_SOL_EJECT_상승 *)
    S369UD_SOL_EJECT_하강 : BOOL; (* AT %MW96423.1 *) (* S369UD_SOL_EJECT_하강 *)
    S369_M_LD_EJECT_상승_LAMP : WORD; (* AT %MW14100 *) (* S369_M_LD_EJECT_상승_LAMP *)
    S369_M_LD_EJECT_하강_LAMP : WORD; (* AT %MW14101 *) (* S369_M_LD_EJECT_하강_LAMP *)
    S369_M_LD_LH_LAT_전진_LAMP : WORD; (* AT %MW14102 *) (* S369_M_LD_LH_LAT_전진_LAMP *)
    S369_M_LD_LH_LAT_후진_LAMP : WORD; (* AT %MW14103 *) (* S369_M_LD_LH_LAT_후진_LAMP *)
    S369_M_LD_RH_LAT_전진_LAMP : WORD; (* AT %MW14104 *) (* S369_M_LD_RH_LAT_전진_LAMP *)
    S369_M_LD_RH_LAT_후진_LAMP : WORD; (* AT %MW14105 *) (* S369_M_LD_RH_LAT_후진_LAMP *)
    S369_M_UD_DOCK_CLP_전진_LAMP : WORD; (* AT %MW14122 *) (* S369_M_UD_DOCK_CLP_전진_LAMP *)
    S369_M_UD_DOCK_CLP_후진_LAMP : WORD; (* AT %MW14123 *) (* S369_M_UD_DOCK_CLP_후진_LAMP *)
    S369_M_UD_EJECT_상승_LAMP : WORD; (* AT %MW14116 *) (* S369_M_UD_EJECT_상승_LAMP *)
    S369_M_UD_EJECT_하강_LAMP : WORD; (* AT %MW14117 *) (* S369_M_UD_EJECT_하강_LAMP *)
    S369_M_UD_LH_LAT_전진_LAMP : WORD; (* AT %MW14118 *) (* S369_M_UD_LH_LAT_전진_LAMP *)
    S369_M_UD_LH_LAT_후진_LAMP : WORD; (* AT %MW14119 *) (* S369_M_UD_LH_LAT_후진_LAMP *)
    S369_M_UD_RH_LAT_전진_LAMP : WORD; (* AT %MW14120 *) (* S369_M_UD_RH_LAT_전진_LAMP *)
    S369_M_UD_RH_LAT_후진_LAMP : WORD; (* AT %MW14121 *) (* S369_M_UD_RH_LAT_후진_LAMP *)
END_VAR
VAR
    S369_LOAD_EJECT : ACT_6_CYL;
    S369_LOAD_LH_LATCH : ACT_6_CYL;
    S369_LOAD_RH_LATCH : ACT_6_CYL;
    S369_UNLOAD_DOCK_CLP : ACT_6_CYL;
    S369_UNLOAD_EJECT : ACT_6_CYL;
    S369_UNLOAD_LH_LATCH : ACT_6_CYL;
    S369_UNLOAD_RH_LATCH : ACT_6_CYL;
END_VAR

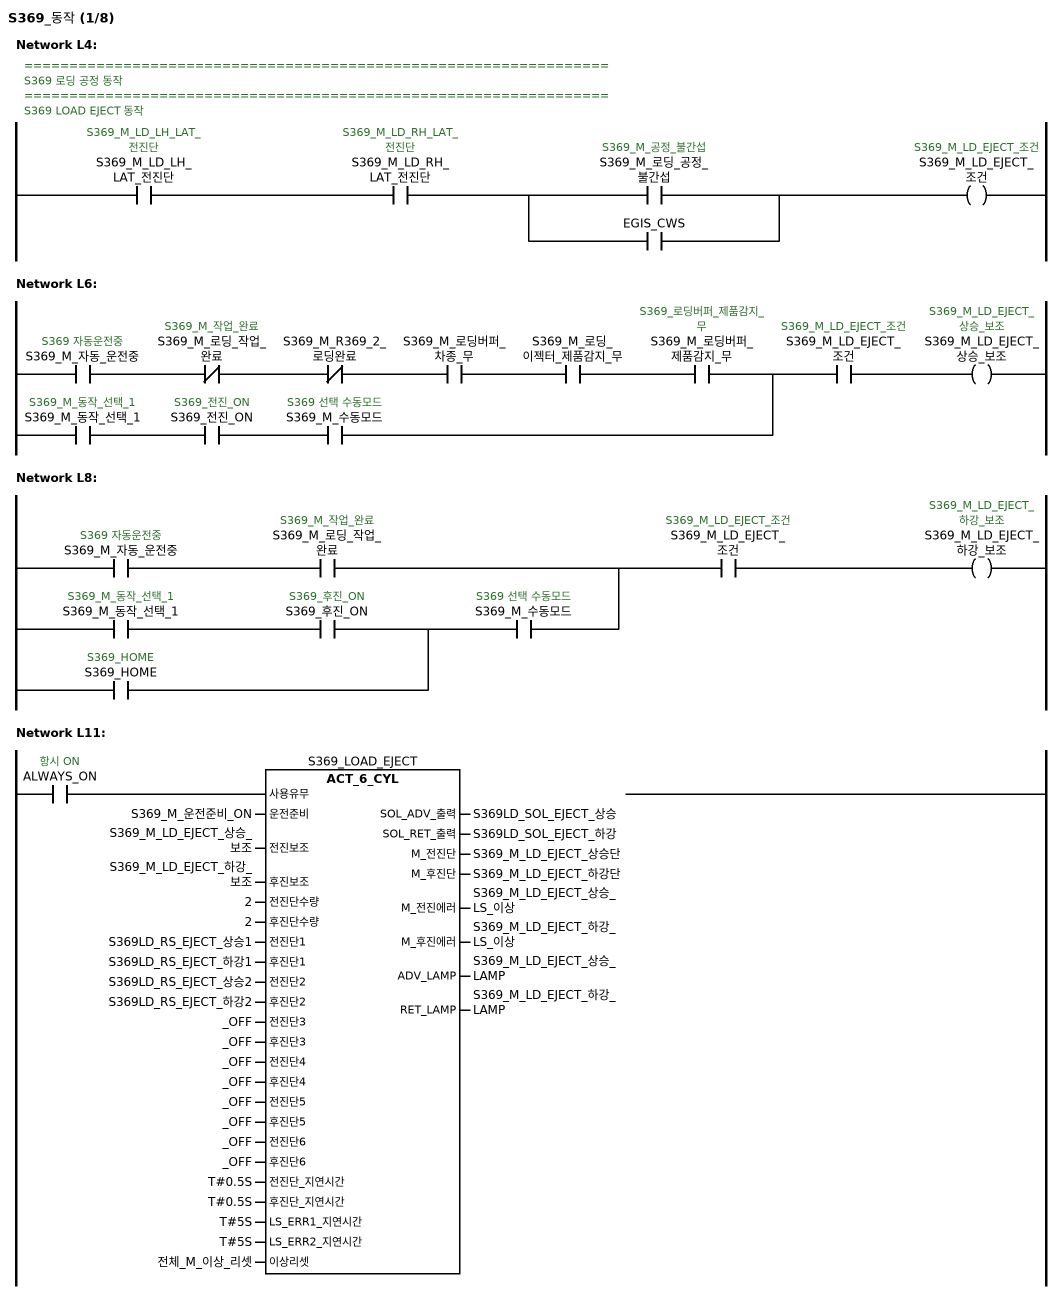
(* ================================================================= *)
(* S369 로딩 공정 동작 *)
(* ================================================================= *)
(* S369 LOAD EJECT 동작 *)
(* Rung L4 *)
S369_M_LD_EJECT_조건 := S369_M_LD_LH_LAT_전진단 AND S369_M_LD_RH_LAT_전진단 AND (S369_M_로딩_공정_불간섭 OR EGIS_CWS);
(* Rung L6 *)
S369_M_LD_EJECT_상승_보조 := ((S369_M_자동_운전중 AND NOT S369_M_로딩_작업_완료 AND NOT S369_M_R369_2_로딩완료 AND S369_M_로딩버퍼_차종_무 AND S369_M_로딩_이젝터_제품감지_무 AND S369_M_로딩버퍼_제품감지_무) OR (S369_M_동작_선택_1 AND S369_전진_ON AND S369_M_수동모드)) AND S369_M_LD_EJECT_조건;
(* Rung L8 *)
S369_M_LD_EJECT_하강_보조 := ((S369_M_자동_운전중 AND S369_M_로딩_작업_완료) OR (((S369_M_동작_선택_1 AND S369_후진_ON) OR S369_HOME) AND S369_M_수동모드)) AND S369_M_LD_EJECT_조건;
(* Rung L11 *)
S369_LOAD_EJECT(사용유무 := ALWAYS_ON, 운전준비 := S369_M_운전준비_ON, 전진보조 := S369_M_LD_EJECT_상승_보조, 후진보조 := S369_M_LD_EJECT_하강_보조, 전진단수량 := 2, 후진단수량 := 2, 전진단1 := S369LD_RS_EJECT_상승1, 후진단1 := S369LD_RS_EJECT_하강1, 전진단2 := S369LD_RS_EJECT_상승2, 후진단2 := S369LD_RS_EJECT_하강2, 전진단3 := _OFF, 후진단3 := _OFF, 전진단4 := _OFF, 후진단4 := _OFF, 전진단5 := _OFF, 후진단5 := _OFF, 전진단6 := _OFF, 후진단6 := _OFF, 전진단_지연시간 := T#0.5S, 후진단_지연시간 := T#0.5S, LS_ERR1_지연시간 := T#5S, LS_ERR2_지연시간 := T#5S, 이상리셋 := 전체_M_이상_리셋, SOL_ADV_출력 => S369LD_SOL_EJECT_상승, SOL_RET_출력 => S369LD_SOL_EJECT_하강, M_전진단 => S369_M_LD_EJECT_상승단, M_후진단 => S369_M_LD_EJECT_하강단, M_전진에러 => S369_M_LD_EJECT_상승_LS_이상, M_후진에러 => S369_M_LD_EJECT_하강_LS_이상, ADV_LAMP => S369_M_LD_EJECT_상승_LAMP, RET_LAMP => S369_M_LD_EJECT_하강_LAMP);

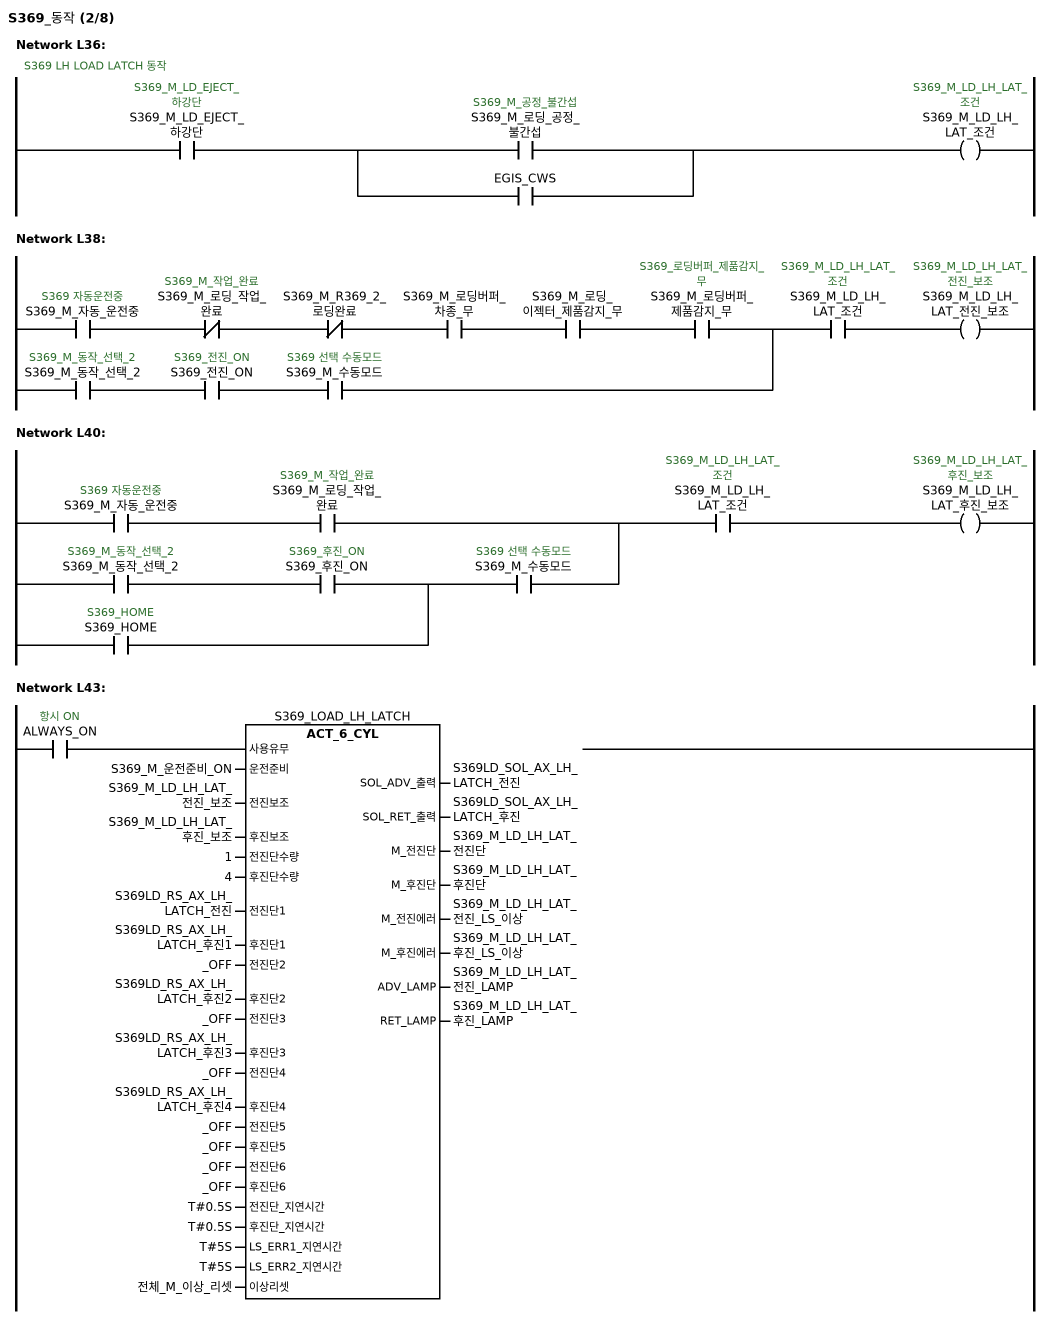
(* S369 LH LOAD LATCH 동작 *)
(* Rung L36 *)
S369_M_LD_LH_LAT_조건 := S369_M_LD_EJECT_하강단 AND (S369_M_로딩_공정_불간섭 OR EGIS_CWS);
(* Rung L38 *)
S369_M_LD_LH_LAT_전진_보조 := ((S369_M_자동_운전중 AND NOT S369_M_로딩_작업_완료 AND NOT S369_M_R369_2_로딩완료 AND S369_M_로딩버퍼_차종_무 AND S369_M_로딩_이젝터_제품감지_무 AND S369_M_로딩버퍼_제품감지_무) OR (S369_M_동작_선택_2 AND S369_전진_ON AND S369_M_수동모드)) AND S369_M_LD_LH_LAT_조건;
(* Rung L40 *)
S369_M_LD_LH_LAT_후진_보조 := ((S369_M_자동_운전중 AND S369_M_로딩_작업_완료) OR (((S369_M_동작_선택_2 AND S369_후진_ON) OR S369_HOME) AND S369_M_수동모드)) AND S369_M_LD_LH_LAT_조건;
(* Rung L43 *)
S369_LOAD_LH_LATCH(사용유무 := ALWAYS_ON, 운전준비 := S369_M_운전준비_ON, 전진보조 := S369_M_LD_LH_LAT_전진_보조, 후진보조 := S369_M_LD_LH_LAT_후진_보조, 전진단수량 := 1, 후진단수량 := 4, 전진단1 := S369LD_RS_AX_LH_LATCH_전진, 후진단1 := S369LD_RS_AX_LH_LATCH_후진1, 전진단2 := _OFF, 후진단2 := S369LD_RS_AX_LH_LATCH_후진2, 전진단3 := _OFF, 후진단3 := S369LD_RS_AX_LH_LATCH_후진3, 전진단4 := _OFF, 후진단4 := S369LD_RS_AX_LH_LATCH_후진4, 전진단5 := _OFF, 후진단5 := _OFF, 전진단6 := _OFF, 후진단6 := _OFF, 전진단_지연시간 := T#0.5S, 후진단_지연시간 := T#0.5S, LS_ERR1_지연시간 := T#5S, LS_ERR2_지연시간 := T#5S, 이상리셋 := 전체_M_이상_리셋, SOL_ADV_출력 => S369LD_SOL_AX_LH_LATCH_전진, SOL_RET_출력 => S369LD_SOL_AX_LH_LATCH_후진, M_전진단 => S369_M_LD_LH_LAT_전진단, M_후진단 => S369_M_LD_LH_LAT_후진단, M_전진에러 => S369_M_LD_LH_LAT_전진_LS_이상, M_후진에러 => S369_M_LD_LH_LAT_후진_LS_이상, ADV_LAMP => S369_M_LD_LH_LAT_전진_LAMP, RET_LAMP => S369_M_LD_LH_LAT_후진_LAMP);

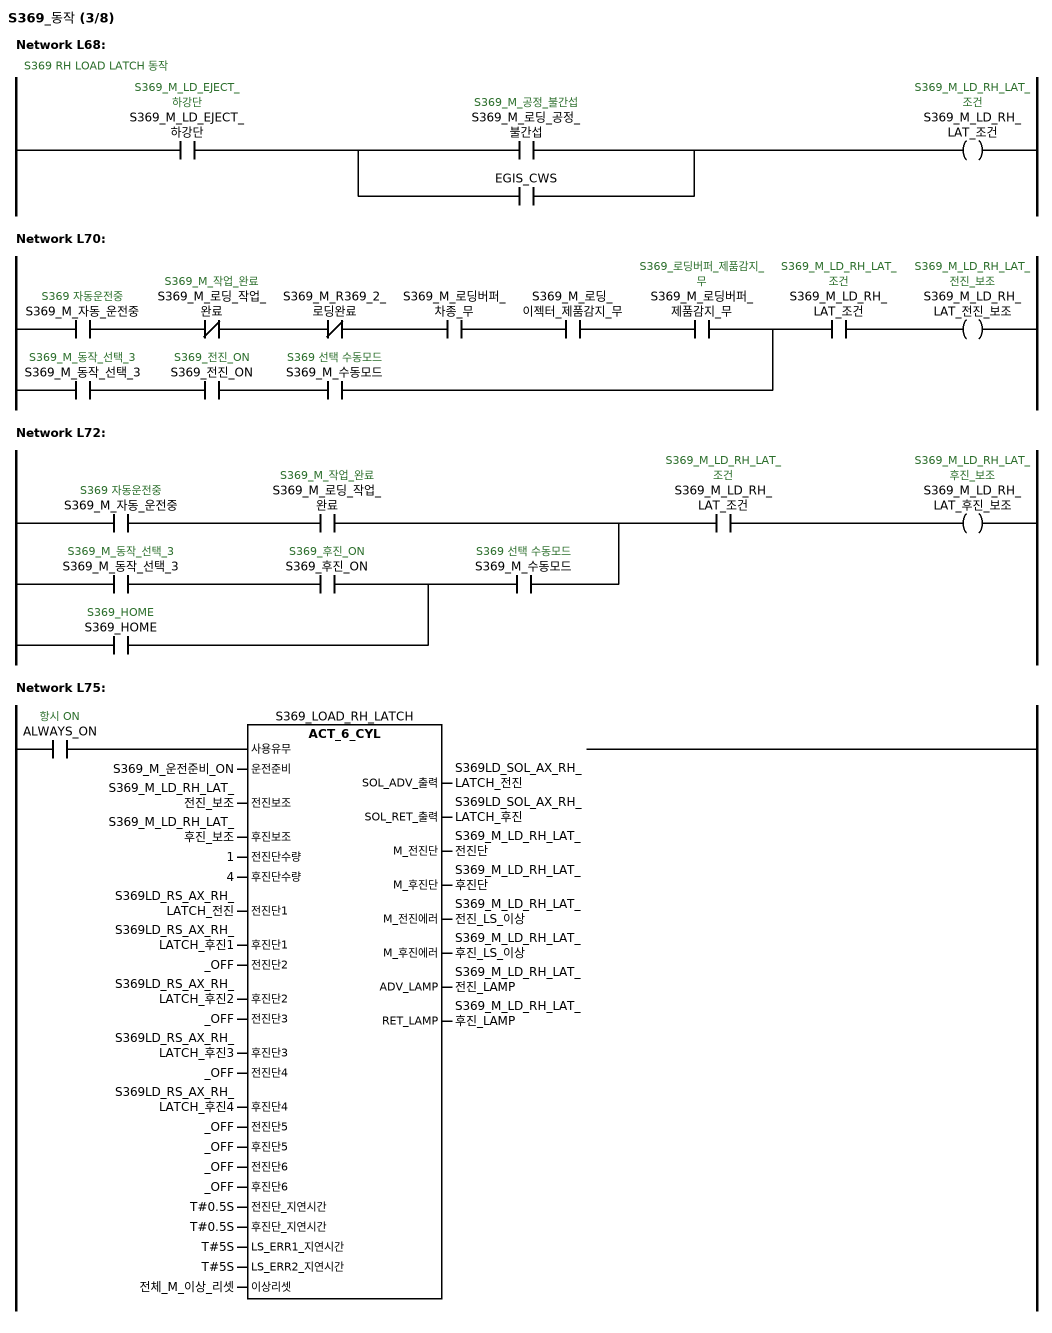
(* S369 RH LOAD LATCH 동작 *)
(* Rung L68 *)
S369_M_LD_RH_LAT_조건 := S369_M_LD_EJECT_하강단 AND (S369_M_로딩_공정_불간섭 OR EGIS_CWS);
(* Rung L70 *)
S369_M_LD_RH_LAT_전진_보조 := ((S369_M_자동_운전중 AND NOT S369_M_로딩_작업_완료 AND NOT S369_M_R369_2_로딩완료 AND S369_M_로딩버퍼_차종_무 AND S369_M_로딩_이젝터_제품감지_무 AND S369_M_로딩버퍼_제품감지_무) OR (S369_M_동작_선택_3 AND S369_전진_ON AND S369_M_수동모드)) AND S369_M_LD_RH_LAT_조건;
(* Rung L72 *)
S369_M_LD_RH_LAT_후진_보조 := ((S369_M_자동_운전중 AND S369_M_로딩_작업_완료) OR (((S369_M_동작_선택_3 AND S369_후진_ON) OR S369_HOME) AND S369_M_수동모드)) AND S369_M_LD_RH_LAT_조건;
(* Rung L75 *)
S369_LOAD_RH_LATCH(사용유무 := ALWAYS_ON, 운전준비 := S369_M_운전준비_ON, 전진보조 := S369_M_LD_RH_LAT_전진_보조, 후진보조 := S369_M_LD_RH_LAT_후진_보조, 전진단수량 := 1, 후진단수량 := 4, 전진단1 := S369LD_RS_AX_RH_LATCH_전진, 후진단1 := S369LD_RS_AX_RH_LATCH_후진1, 전진단2 := _OFF, 후진단2 := S369LD_RS_AX_RH_LATCH_후진2, 전진단3 := _OFF, 후진단3 := S369LD_RS_AX_RH_LATCH_후진3, 전진단4 := _OFF, 후진단4 := S369LD_RS_AX_RH_LATCH_후진4, 전진단5 := _OFF, 후진단5 := _OFF, 전진단6 := _OFF, 후진단6 := _OFF, 전진단_지연시간 := T#0.5S, 후진단_지연시간 := T#0.5S, LS_ERR1_지연시간 := T#5S, LS_ERR2_지연시간 := T#5S, 이상리셋 := 전체_M_이상_리셋, SOL_ADV_출력 => S369LD_SOL_AX_RH_LATCH_전진, SOL_RET_출력 => S369LD_SOL_AX_RH_LATCH_후진, M_전진단 => S369_M_LD_RH_LAT_전진단, M_후진단 => S369_M_LD_RH_LAT_후진단, M_전진에러 => S369_M_LD_RH_LAT_전진_LS_이상, M_후진에러 => S369_M_LD_RH_LAT_후진_LS_이상, ADV_LAMP => S369_M_LD_RH_LAT_전진_LAMP, RET_LAMP => S369_M_LD_RH_LAT_후진_LAMP);

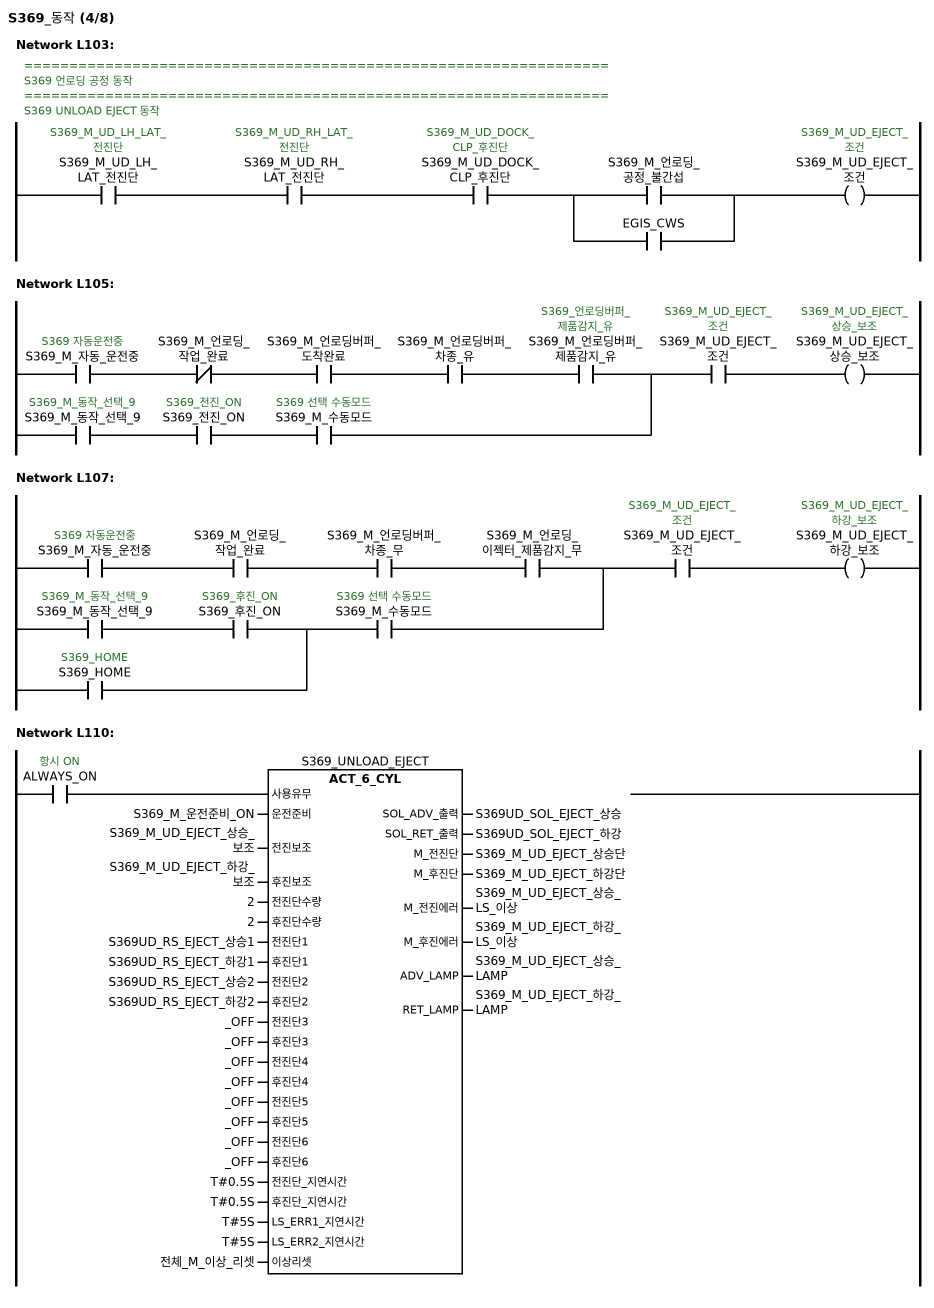
(* ================================================================= *)
(* S369 언로딩 공정 동작 *)
(* ================================================================= *)
(* S369 UNLOAD EJECT 동작 *)
(* Rung L103 *)
S369_M_UD_EJECT_조건 := S369_M_UD_LH_LAT_전진단 AND S369_M_UD_RH_LAT_전진단 AND S369_M_UD_DOCK_CLP_후진단 AND (S369_M_언로딩_공정_불간섭 OR EGIS_CWS);
(* Rung L105 *)
S369_M_UD_EJECT_상승_보조 := ((S369_M_자동_운전중 AND NOT S369_M_언로딩_작업_완료 AND S369_M_언로딩버퍼_도착완료 AND S369_M_언로딩버퍼_차종_유 AND S369_M_언로딩버퍼_제품감지_유) OR (S369_M_동작_선택_9 AND S369_전진_ON AND S369_M_수동모드)) AND S369_M_UD_EJECT_조건;
(* Rung L107 *)
S369_M_UD_EJECT_하강_보조 := ((S369_M_자동_운전중 AND S369_M_언로딩_작업_완료 AND S369_M_언로딩버퍼_차종_무 AND S369_M_언로딩_이젝터_제품감지_무) OR (((S369_M_동작_선택_9 AND S369_후진_ON) OR S369_HOME) AND S369_M_수동모드)) AND S369_M_UD_EJECT_조건;
(* Rung L110 *)
S369_UNLOAD_EJECT(사용유무 := ALWAYS_ON, 운전준비 := S369_M_운전준비_ON, 전진보조 := S369_M_UD_EJECT_상승_보조, 후진보조 := S369_M_UD_EJECT_하강_보조, 전진단수량 := 2, 후진단수량 := 2, 전진단1 := S369UD_RS_EJECT_상승1, 후진단1 := S369UD_RS_EJECT_하강1, 전진단2 := S369UD_RS_EJECT_상승2, 후진단2 := S369UD_RS_EJECT_하강2, 전진단3 := _OFF, 후진단3 := _OFF, 전진단4 := _OFF, 후진단4 := _OFF, 전진단5 := _OFF, 후진단5 := _OFF, 전진단6 := _OFF, 후진단6 := _OFF, 전진단_지연시간 := T#0.5S, 후진단_지연시간 := T#0.5S, LS_ERR1_지연시간 := T#5S, LS_ERR2_지연시간 := T#5S, 이상리셋 := 전체_M_이상_리셋, SOL_ADV_출력 => S369UD_SOL_EJECT_상승, SOL_RET_출력 => S369UD_SOL_EJECT_하강, M_전진단 => S369_M_UD_EJECT_상승단, M_후진단 => S369_M_UD_EJECT_하강단, M_전진에러 => S369_M_UD_EJECT_상승_LS_이상, M_후진에러 => S369_M_UD_EJECT_하강_LS_이상, ADV_LAMP => S369_M_UD_EJECT_상승_LAMP, RET_LAMP => S369_M_UD_EJECT_하강_LAMP);

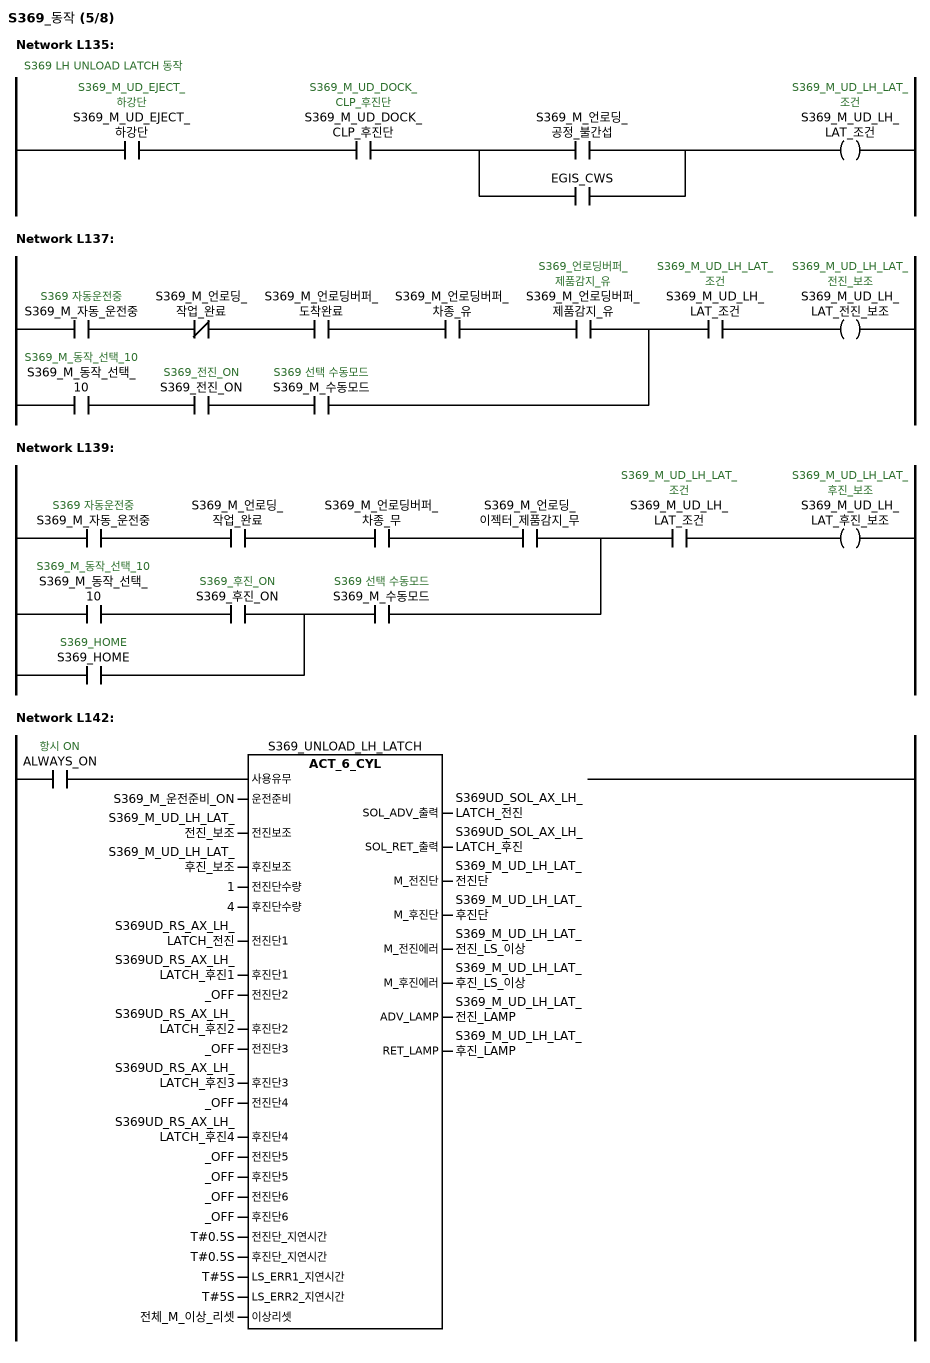
(* S369 LH UNLOAD LATCH 동작 *)
(* Rung L135 *)
S369_M_UD_LH_LAT_조건 := S369_M_UD_EJECT_하강단 AND S369_M_UD_DOCK_CLP_후진단 AND (S369_M_언로딩_공정_불간섭 OR EGIS_CWS);
(* Rung L137 *)
S369_M_UD_LH_LAT_전진_보조 := ((S369_M_자동_운전중 AND NOT S369_M_언로딩_작업_완료 AND S369_M_언로딩버퍼_도착완료 AND S369_M_언로딩버퍼_차종_유 AND S369_M_언로딩버퍼_제품감지_유) OR (S369_M_동작_선택_10 AND S369_전진_ON AND S369_M_수동모드)) AND S369_M_UD_LH_LAT_조건;
(* Rung L139 *)
S369_M_UD_LH_LAT_후진_보조 := ((S369_M_자동_운전중 AND S369_M_언로딩_작업_완료 AND S369_M_언로딩버퍼_차종_무 AND S369_M_언로딩_이젝터_제품감지_무) OR (((S369_M_동작_선택_10 AND S369_후진_ON) OR S369_HOME) AND S369_M_수동모드)) AND S369_M_UD_LH_LAT_조건;
(* Rung L142 *)
S369_UNLOAD_LH_LATCH(사용유무 := ALWAYS_ON, 운전준비 := S369_M_운전준비_ON, 전진보조 := S369_M_UD_LH_LAT_전진_보조, 후진보조 := S369_M_UD_LH_LAT_후진_보조, 전진단수량 := 1, 후진단수량 := 4, 전진단1 := S369UD_RS_AX_LH_LATCH_전진, 후진단1 := S369UD_RS_AX_LH_LATCH_후진1, 전진단2 := _OFF, 후진단2 := S369UD_RS_AX_LH_LATCH_후진2, 전진단3 := _OFF, 후진단3 := S369UD_RS_AX_LH_LATCH_후진3, 전진단4 := _OFF, 후진단4 := S369UD_RS_AX_LH_LATCH_후진4, 전진단5 := _OFF, 후진단5 := _OFF, 전진단6 := _OFF, 후진단6 := _OFF, 전진단_지연시간 := T#0.5S, 후진단_지연시간 := T#0.5S, LS_ERR1_지연시간 := T#5S, LS_ERR2_지연시간 := T#5S, 이상리셋 := 전체_M_이상_리셋, SOL_ADV_출력 => S369UD_SOL_AX_LH_LATCH_전진, SOL_RET_출력 => S369UD_SOL_AX_LH_LATCH_후진, M_전진단 => S369_M_UD_LH_LAT_전진단, M_후진단 => S369_M_UD_LH_LAT_후진단, M_전진에러 => S369_M_UD_LH_LAT_전진_LS_이상, M_후진에러 => S369_M_UD_LH_LAT_후진_LS_이상, ADV_LAMP => S369_M_UD_LH_LAT_전진_LAMP, RET_LAMP => S369_M_UD_LH_LAT_후진_LAMP);

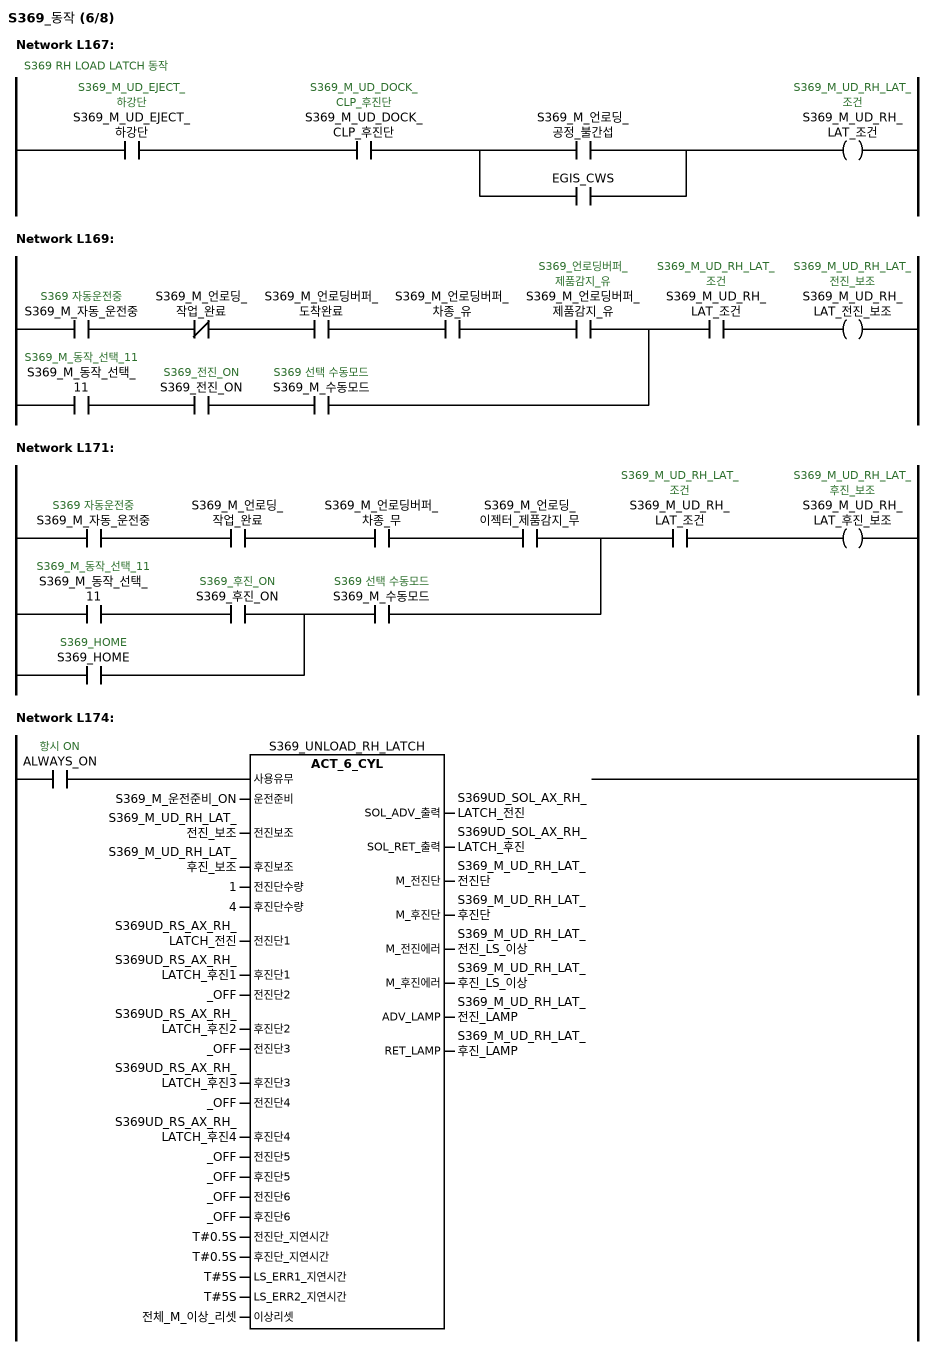
(* S369 RH LOAD LATCH 동작 *)
(* Rung L167 *)
S369_M_UD_RH_LAT_조건 := S369_M_UD_EJECT_하강단 AND S369_M_UD_DOCK_CLP_후진단 AND (S369_M_언로딩_공정_불간섭 OR EGIS_CWS);
(* Rung L169 *)
S369_M_UD_RH_LAT_전진_보조 := ((S369_M_자동_운전중 AND NOT S369_M_언로딩_작업_완료 AND S369_M_언로딩버퍼_도착완료 AND S369_M_언로딩버퍼_차종_유 AND S369_M_언로딩버퍼_제품감지_유) OR (S369_M_동작_선택_11 AND S369_전진_ON AND S369_M_수동모드)) AND S369_M_UD_RH_LAT_조건;
(* Rung L171 *)
S369_M_UD_RH_LAT_후진_보조 := ((S369_M_자동_운전중 AND S369_M_언로딩_작업_완료 AND S369_M_언로딩버퍼_차종_무 AND S369_M_언로딩_이젝터_제품감지_무) OR (((S369_M_동작_선택_11 AND S369_후진_ON) OR S369_HOME) AND S369_M_수동모드)) AND S369_M_UD_RH_LAT_조건;
(* Rung L174 *)
S369_UNLOAD_RH_LATCH(사용유무 := ALWAYS_ON, 운전준비 := S369_M_운전준비_ON, 전진보조 := S369_M_UD_RH_LAT_전진_보조, 후진보조 := S369_M_UD_RH_LAT_후진_보조, 전진단수량 := 1, 후진단수량 := 4, 전진단1 := S369UD_RS_AX_RH_LATCH_전진, 후진단1 := S369UD_RS_AX_RH_LATCH_후진1, 전진단2 := _OFF, 후진단2 := S369UD_RS_AX_RH_LATCH_후진2, 전진단3 := _OFF, 후진단3 := S369UD_RS_AX_RH_LATCH_후진3, 전진단4 := _OFF, 후진단4 := S369UD_RS_AX_RH_LATCH_후진4, 전진단5 := _OFF, 후진단5 := _OFF, 전진단6 := _OFF, 후진단6 := _OFF, 전진단_지연시간 := T#0.5S, 후진단_지연시간 := T#0.5S, LS_ERR1_지연시간 := T#5S, LS_ERR2_지연시간 := T#5S, 이상리셋 := 전체_M_이상_리셋, SOL_ADV_출력 => S369UD_SOL_AX_RH_LATCH_전진, SOL_RET_출력 => S369UD_SOL_AX_RH_LATCH_후진, M_전진단 => S369_M_UD_RH_LAT_전진단, M_후진단 => S369_M_UD_RH_LAT_후진단, M_전진에러 => S369_M_UD_RH_LAT_전진_LS_이상, M_후진에러 => S369_M_UD_RH_LAT_후진_LS_이상, ADV_LAMP => S369_M_UD_RH_LAT_전진_LAMP, RET_LAMP => S369_M_UD_RH_LAT_후진_LAMP);

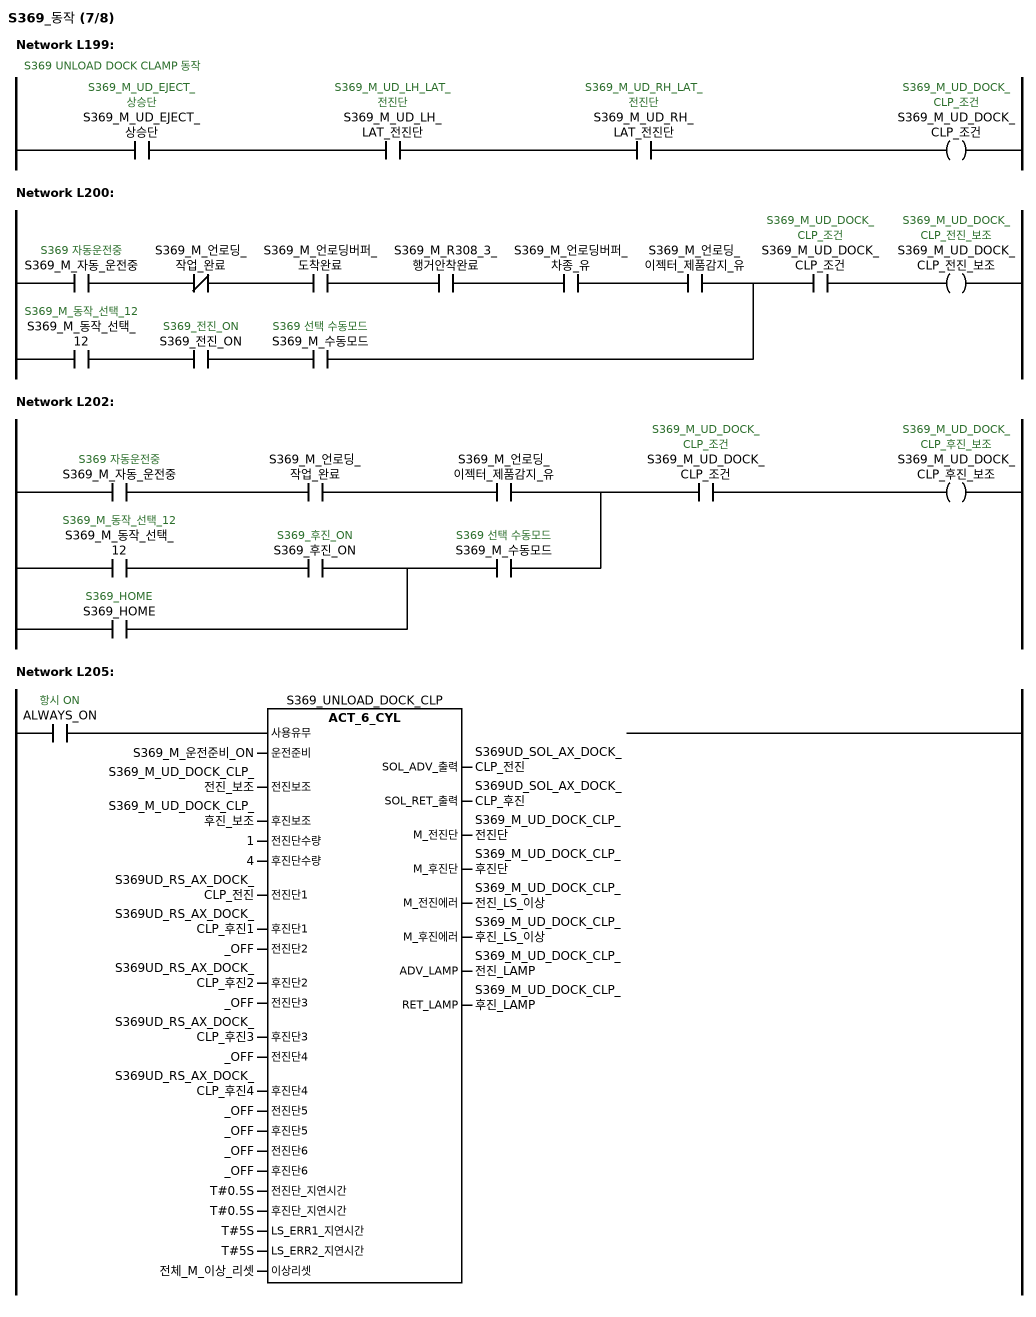
(* S369 UNLOAD DOCK CLAMP 동작 *)
(* Rung L199 *)
S369_M_UD_DOCK_CLP_조건 := S369_M_UD_EJECT_상승단 AND S369_M_UD_LH_LAT_전진단 AND S369_M_UD_RH_LAT_전진단;
(* Rung L200 *)
S369_M_UD_DOCK_CLP_전진_보조 := ((S369_M_자동_운전중 AND NOT S369_M_언로딩_작업_완료 AND S369_M_언로딩버퍼_도착완료 AND S369_M_R308_3_행거안착완료 AND S369_M_언로딩버퍼_차종_유 AND S369_M_언로딩_이젝터_제품감지_유) OR (S369_M_동작_선택_12 AND S369_전진_ON AND S369_M_수동모드)) AND S369_M_UD_DOCK_CLP_조건;
(* Rung L202 *)
S369_M_UD_DOCK_CLP_후진_보조 := ((S369_M_자동_운전중 AND S369_M_언로딩_작업_완료 AND S369_M_언로딩_이젝터_제품감지_유) OR (((S369_M_동작_선택_12 AND S369_후진_ON) OR S369_HOME) AND S369_M_수동모드)) AND S369_M_UD_DOCK_CLP_조건;
(* Rung L205 *)
S369_UNLOAD_DOCK_CLP(사용유무 := ALWAYS_ON, 운전준비 := S369_M_운전준비_ON, 전진보조 := S369_M_UD_DOCK_CLP_전진_보조, 후진보조 := S369_M_UD_DOCK_CLP_후진_보조, 전진단수량 := 1, 후진단수량 := 4, 전진단1 := S369UD_RS_AX_DOCK_CLP_전진, 후진단1 := S369UD_RS_AX_DOCK_CLP_후진1, 전진단2 := _OFF, 후진단2 := S369UD_RS_AX_DOCK_CLP_후진2, 전진단3 := _OFF, 후진단3 := S369UD_RS_AX_DOCK_CLP_후진3, 전진단4 := _OFF, 후진단4 := S369UD_RS_AX_DOCK_CLP_후진4, 전진단5 := _OFF, 후진단5 := _OFF, 전진단6 := _OFF, 후진단6 := _OFF, 전진단_지연시간 := T#0.5S, 후진단_지연시간 := T#0.5S, LS_ERR1_지연시간 := T#5S, LS_ERR2_지연시간 := T#5S, 이상리셋 := 전체_M_이상_리셋, SOL_ADV_출력 => S369UD_SOL_AX_DOCK_CLP_전진, SOL_RET_출력 => S369UD_SOL_AX_DOCK_CLP_후진, M_전진단 => S369_M_UD_DOCK_CLP_전진단, M_후진단 => S369_M_UD_DOCK_CLP_후진단, M_전진에러 => S369_M_UD_DOCK_CLP_전진_LS_이상, M_후진에러 => S369_M_UD_DOCK_CLP_후진_LS_이상, ADV_LAMP => S369_M_UD_DOCK_CLP_전진_LAMP, RET_LAMP => S369_M_UD_DOCK_CLP_후진_LAMP);

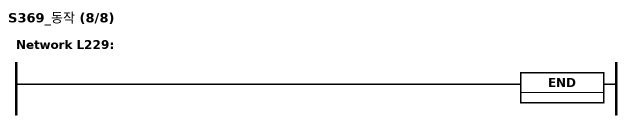
(* Rung L229 *)
END();
END_PROGRAM

PROGRAM S369_외부설비(컨베어_이송장치) (* task: 스캔 프로그램 *)
VAR_EXTERNAL RETAIN
    ALWAYS_OFF : BOOL; (* AT %MW3.0 *) (* 항시 OFF *)
    ALWAYS_ON : BOOL; (* AT %MW3.1 *) (* 항시 ON *)
    S369_M_동작_선택_8 : BOOL; (* AT %MW5040.7 *) (* S369_M_동작_선택_8 *)
    S369_M_로딩_공정_원위치 : BOOL; (* AT %MW5004.0 *) (* S369_M_공정_원위치 *)
    S369_M_로딩_리셋보조 : BOOL; (* AT %MW5000.13 *)
    S369_M_로딩_작업_완료 : BOOL; (* AT %MW5001.0 *) (* S369_M_작업_완료 *)
    S369_M_수동모드 : BOOL; (* AT %MW5000.3 *) (* S369 선택 수동모드 *)
    S369_M_언로딩_공정_원위치 : BOOL; (* AT %MW5004.1 *)
    S369_M_언로딩_이젝터_제품감지_무 : BOOL; (* AT %MW5001.11 *)
    S369_M_언로딩_작업_완료 : BOOL; (* AT %MW5001.1 *)
    S369_M_언로딩버퍼_도착완료 : BOOL; (* AT %MW5003.6 *)
    S369_M_언로딩버퍼_제품감지_무 : BOOL; (* AT %MW5005.11 *) (* S369_언로딩버퍼_제품감지_무 *)
    S369_M_언로딩버퍼_제품감지_유 : BOOL; (* AT %MW5005.10 *) (* S369_언로딩버퍼_제품감지_유 *)
    S369_M_언로딩버퍼_차종_무 : BOOL; (* AT %MW5002.3 *)
    S369_M_언로딩버퍼_차종_유 : BOOL; (* AT %MW5002.2 *)
    S369_M_운전준비_ON : BOOL; (* AT %MW5000.0 *) (* S369 운전준비 ON *)
    S369_M_이송버퍼01_제품감지_유 : BOOL; (* AT %MW5005.8 *) (* S369_이송버퍼01_제품감지_ON *)
    S369_M_이송버퍼02_제품감지_유 : BOOL; (* AT %MW5005.6 *) (* S369_이송버퍼02_제품감지_ON *)
    S369_M_이송버퍼03_제품감지_유 : BOOL; (* AT %MW5005.4 *) (* S369_이송버퍼03_제품감지_ON *)
    S369_M_이송버퍼04_제품감지_유 : BOOL; (* AT %MW5005.2 *) (* S369_이송버퍼04_제품감지_ON *)
    S369_M_이송버퍼1_도착완료 : BOOL; (* AT %MW5003.5 *)
    S369_M_이송버퍼1_차종_무 : BOOL; (* AT %MW5002.11 *)
    S369_M_이송버퍼1_차종_유 : BOOL; (* AT %MW5002.10 *)
    S369_M_이송버퍼2_도착완료 : BOOL; (* AT %MW5003.4 *)
    S369_M_이송버퍼2_차종_무 : BOOL; (* AT %MW5002.9 *)
    S369_M_이송버퍼2_차종_유 : BOOL; (* AT %MW5002.8 *)
    S369_M_이송버퍼3_도착완료 : BOOL; (* AT %MW5003.3 *)
    S369_M_이송버퍼3_차종_무 : BOOL; (* AT %MW5002.7 *)
    S369_M_이송버퍼3_차종_유 : BOOL; (* AT %MW5002.6 *)
    S369_M_이송버퍼4_도착완료 : BOOL; (* AT %MW5003.2 *)
    S369_M_이송버퍼4_차종_무 : BOOL; (* AT %MW5002.5 *)
    S369_M_이송버퍼4_차종_유 : BOOL; (* AT %MW5002.4 *)
    S369_M_자동_운전중 : BOOL; (* AT %MW5000.4 *) (* S369 자동운전중 *)
    S369_M_전체_컨베어_도착완료 : BOOL; (* AT %MW5003.0 *)
    S369_M_컨베어_이동가능 : BOOL; (* AT %MW5107.8 *)
    S369_M_컨베어_차종무_도착완료 : BOOL; (* AT %MW5003.1 *)
    S369_M_콘베어_이동_전진_보조 : BOOL; (* AT %MW5107.1 *)
    S369_M_콘베어_이동_조건 : BOOL; (* AT %MW5107.0 *)
    S369_M_콘베어_이동_후진_보조 : BOOL; (* AT %MW5107.2 *)
    S369_전진_ON : BOOL; (* AT %MW5048.1 *) (* S369_전진_ON *)
    S369_후진_ON : BOOL; (* AT %MW5048.2 *) (* S369_후진_ON *)
    전체_M_이상_리셋 : BOOL; (* AT %MW308.2 *) (* ALL공정 PB 이상리셋 *)
END_VAR
VAR
    INST : TP;
    INST1 : TP;
    INST2 : TP;
    INST3 : TP;
    INST4 : TP;
    INST5 : TP;
    INST6 : TON;
END_VAR
VAR_EXTERNAL
    S369_CONVEY_I_모터기동중 : BOOL; (* AT %MW50000.4 *)
    S369_CONVEY_I_서보_운전준비 : BOOL; (* AT %MW50000.0 *)
    S369_CONVEY_O_JERK_LIMIT : DINT; (* AT %MD25014 *)
    S369_CONVEY_O_JOG_모드비활성 : BOOL; (* AT %MW50020.5 *)
    S369_CONVEY_O_JOG_모드활성 : BOOL; (* AT %MW50020.4 *)
    S369_CONVEY_O_가속설정 : UINT; (* AT %MW50022 *)
    S369_CONVEY_O_감속설정 : UINT; (* AT %MW50023 *)
    S369_CONVEY_O_구동모드설정 : UINT; (* AT %MW50025 *)
    S369_CONVEY_O_기동정지 : BOOL; (* AT %MW50020.1 *)
    S369_CONVEY_O_비상정지 : BOOL; (* AT %MW50020.0 *)
    S369_CONVEY_O_이동속도_설정 : UINT; (* AT %MW50021 *)
    S369_CONVEY_O_이상리셋 : BOOL; (* AT %MW50020.8 *)
    SERVO_SAFETY_CR_ON : BOOL; (* AT %MW95024.0 *) (* SERVO_BRAKE_CR_ON *)
END_VAR
VAR
    _e1 : R_TRIG;
    _e2 : R_TRIG;
    _p3 : BOOL;
    _e4 : R_TRIG;
    _p5 : BOOL;
END_VAR

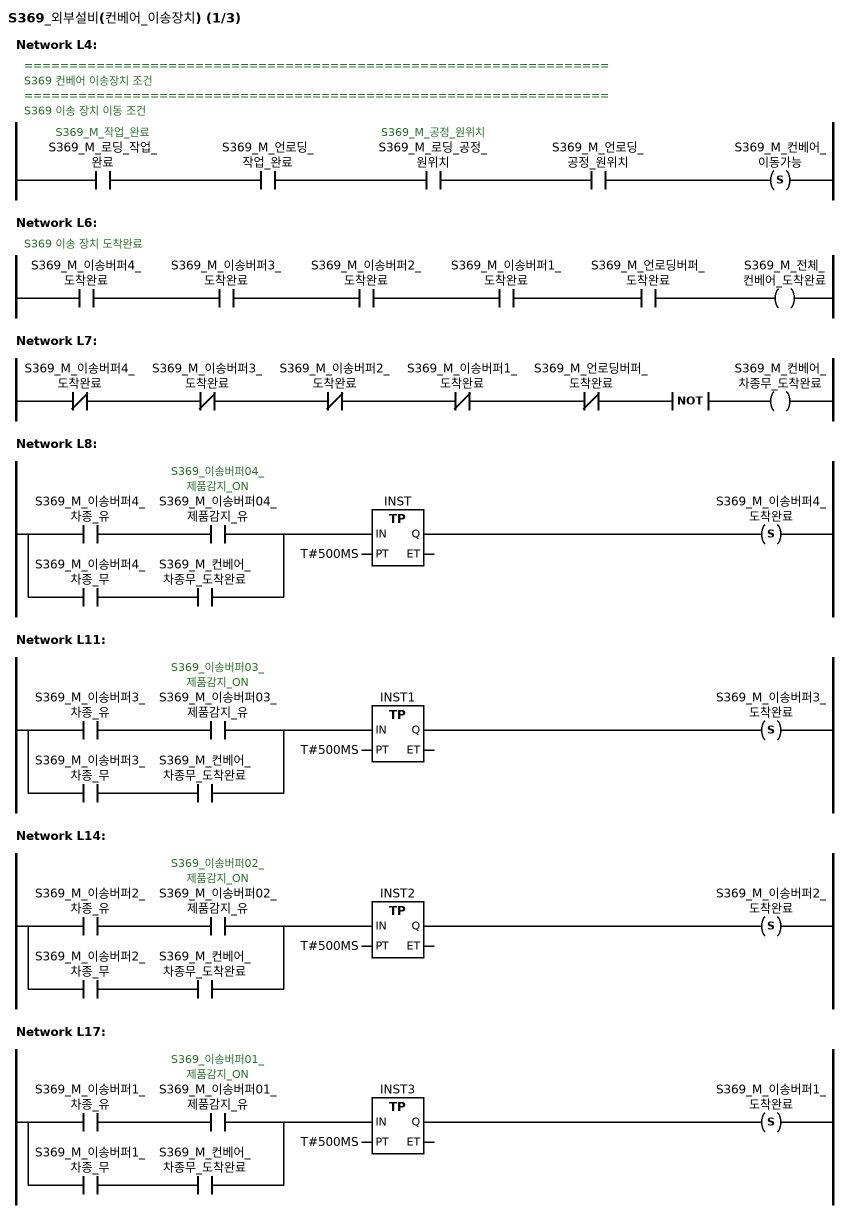
(* ================================================================= *)
(* S369 컨베어 이송장치 조건 *)
(* ================================================================= *)
(* S369 이송 장치 이동 조건 *)
(* Rung L4 *)
IF S369_M_로딩_작업_완료 AND S369_M_언로딩_작업_완료 AND S369_M_로딩_공정_원위치 AND S369_M_언로딩_공정_원위치 THEN
    S369_M_컨베어_이동가능 := TRUE;
END_IF;
(* S369 이송 장치 도착완료 *)
(* Rung L6 *)
S369_M_전체_컨베어_도착완료 := S369_M_이송버퍼4_도착완료 AND S369_M_이송버퍼3_도착완료 AND S369_M_이송버퍼2_도착완료 AND S369_M_이송버퍼1_도착완료 AND S369_M_언로딩버퍼_도착완료;
(* Rung L7 *)
S369_M_컨베어_차종무_도착완료 := NOT (NOT S369_M_이송버퍼4_도착완료 AND NOT S369_M_이송버퍼3_도착완료 AND NOT S369_M_이송버퍼2_도착완료 AND NOT S369_M_이송버퍼1_도착완료 AND NOT S369_M_언로딩버퍼_도착완료);
(* Rung L8 *)
INST(IN := (S369_M_이송버퍼4_차종_유 AND S369_M_이송버퍼04_제품감지_유) OR (S369_M_이송버퍼4_차종_무 AND S369_M_컨베어_차종무_도착완료), PT := T#500MS);
IF INST.Q THEN S369_M_이송버퍼4_도착완료 := TRUE; END_IF;
(* Rung L11 *)
INST1(IN := (S369_M_이송버퍼3_차종_유 AND S369_M_이송버퍼03_제품감지_유) OR (S369_M_이송버퍼3_차종_무 AND S369_M_컨베어_차종무_도착완료), PT := T#500MS);
IF INST1.Q THEN S369_M_이송버퍼3_도착완료 := TRUE; END_IF;
(* Rung L14 *)
INST2(IN := (S369_M_이송버퍼2_차종_유 AND S369_M_이송버퍼02_제품감지_유) OR (S369_M_이송버퍼2_차종_무 AND S369_M_컨베어_차종무_도착완료), PT := T#500MS);
IF INST2.Q THEN S369_M_이송버퍼2_도착완료 := TRUE; END_IF;
(* Rung L17 *)
INST3(IN := (S369_M_이송버퍼1_차종_유 AND S369_M_이송버퍼01_제품감지_유) OR (S369_M_이송버퍼1_차종_무 AND S369_M_컨베어_차종무_도착완료), PT := T#500MS);
IF INST3.Q THEN S369_M_이송버퍼1_도착완료 := TRUE; END_IF;

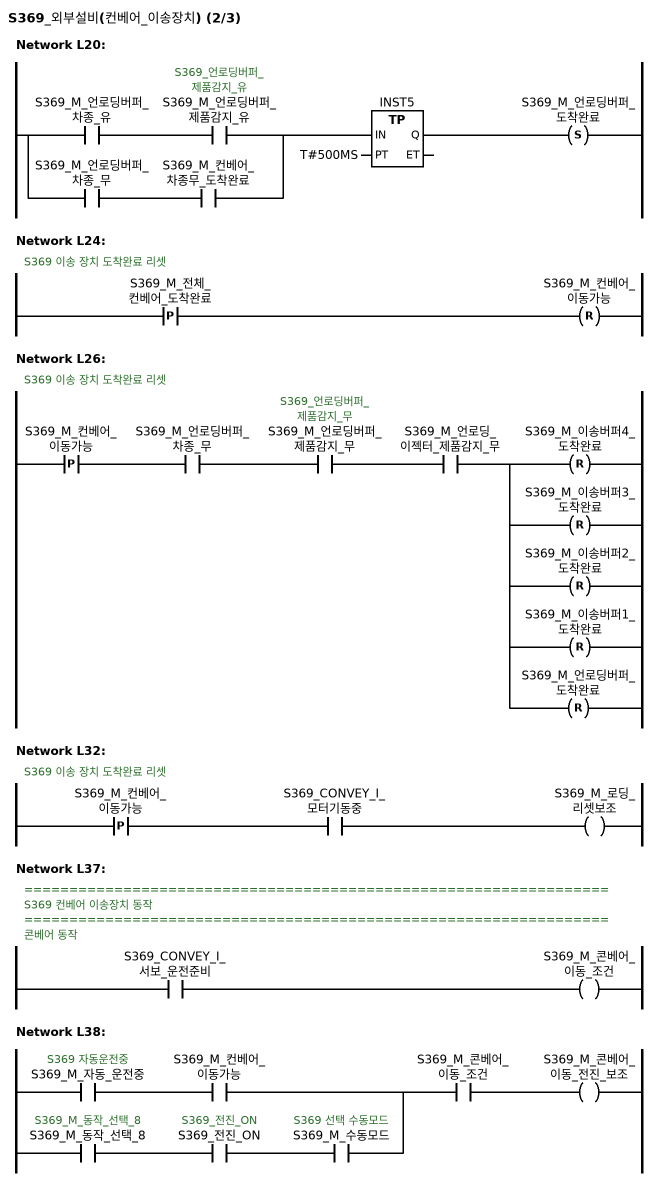
(* Rung L20 *)
INST5(IN := (S369_M_언로딩버퍼_차종_유 AND S369_M_언로딩버퍼_제품감지_유) OR (S369_M_언로딩버퍼_차종_무 AND S369_M_컨베어_차종무_도착완료), PT := T#500MS);
IF INST5.Q THEN S369_M_언로딩버퍼_도착완료 := TRUE; END_IF;
(* S369 이송 장치 도착완료 리셋 *)
(* Rung L24 *)
_e1(CLK := S369_M_전체_컨베어_도착완료);
IF _e1.Q THEN S369_M_컨베어_이동가능 := FALSE; END_IF;
(* S369 이송 장치 도착완료 리셋 *)
(* Rung L26 *)
_e2(CLK := S369_M_컨베어_이동가능);
_p3 := _e2.Q AND S369_M_언로딩버퍼_차종_무 AND S369_M_언로딩버퍼_제품감지_무 AND S369_M_언로딩_이젝터_제품감지_무;
IF _p3 THEN
    S369_M_이송버퍼4_도착완료 := FALSE;
    S369_M_이송버퍼3_도착완료 := FALSE;
    S369_M_이송버퍼2_도착완료 := FALSE;
    S369_M_이송버퍼1_도착완료 := FALSE;
    S369_M_언로딩버퍼_도착완료 := FALSE;
END_IF;
(* S369 이송 장치 도착완료 리셋 *)
(* Rung L32 *)
_e4(CLK := S369_M_컨베어_이동가능);
S369_M_로딩_리셋보조 := _e4.Q AND S369_CONVEY_I_모터기동중;
(* ================================================================= *)
(* S369 컨베어 이송장치 동작 *)
(* ================================================================= *)
(* 콘베어 동작 *)
(* Rung L37 *)
S369_M_콘베어_이동_조건 := S369_CONVEY_I_서보_운전준비;
(* Rung L38 *)
S369_M_콘베어_이동_전진_보조 := ((S369_M_자동_운전중 AND S369_M_컨베어_이동가능) OR (S369_M_동작_선택_8 AND S369_전진_ON AND S369_M_수동모드)) AND S369_M_콘베어_이동_조건;

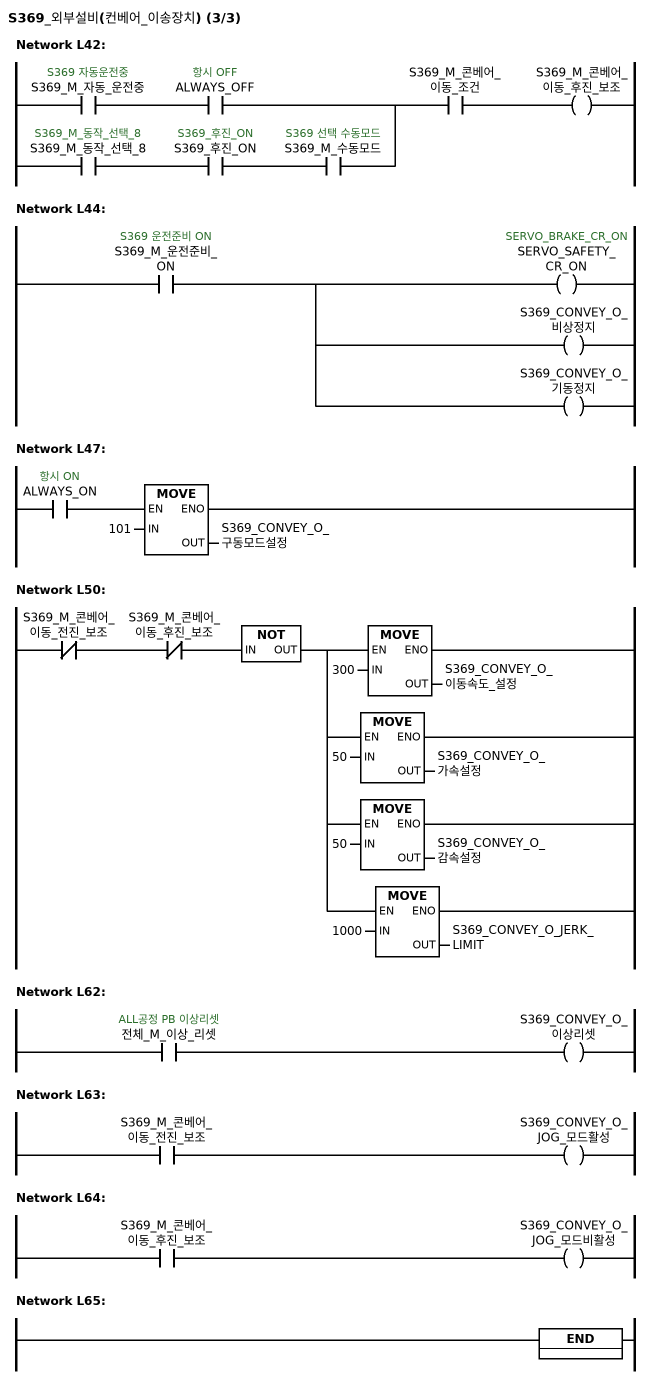
(* Rung L42 *)
S369_M_콘베어_이동_후진_보조 := ((S369_M_자동_운전중 AND ALWAYS_OFF) OR (S369_M_동작_선택_8 AND S369_후진_ON AND S369_M_수동모드)) AND S369_M_콘베어_이동_조건;
(* Rung L44 *)
SERVO_SAFETY_CR_ON := S369_M_운전준비_ON;
S369_CONVEY_O_비상정지 := S369_M_운전준비_ON;
S369_CONVEY_O_기동정지 := S369_M_운전준비_ON;
(* Rung L47 *)
IF ALWAYS_ON THEN S369_CONVEY_O_구동모드설정 := 101; END_IF;
(* Rung L50 *)
_p5 := NOT (NOT S369_M_콘베어_이동_전진_보조 AND NOT S369_M_콘베어_이동_후진_보조);
IF _p5 THEN
    S369_CONVEY_O_이동속도_설정 := 300;
    S369_CONVEY_O_가속설정 := 50;
    S369_CONVEY_O_감속설정 := 50;
    S369_CONVEY_O_JERK_LIMIT := 1000;
END_IF;
(* Rung L62 *)
S369_CONVEY_O_이상리셋 := 전체_M_이상_리셋;
(* Rung L63 *)
S369_CONVEY_O_JOG_모드활성 := S369_M_콘베어_이동_전진_보조;
(* Rung L64 *)
S369_CONVEY_O_JOG_모드비활성 := S369_M_콘베어_이동_후진_보조;
(* Rung L65 *)
END();
END_PROGRAM

PROGRAM S369_인터록 (* task: 스캔 프로그램 *)
VAR_EXTERNAL
    BB_MAIN_I_차종_요구 : BOOL; (* AT %MW83011.3 *)
    BB_MAIN_O_SAFETY_이상 : BOOL; (* AT %MW93010.14 *)
    BB_MAIN_O_불간섭 : BOOL; (* AT %MW93011.0 *)
    BB_MAIN_O_비상정지 : BOOL; (* AT %MW93010.15 *)
    BB_MAIN_O_운전준비 : BOOL; (* AT %MW93010.0 *)
    BB_MAIN_O_이상 : BOOL; (* AT %MW93010.13 *)
    BB_MAIN_O_자동기동 : BOOL; (* AT %MW93010.3 *)
    BB_MAIN_O_진입_OK : BOOL; (* AT %MW93011.1 *)
    BB_MAIN_O_취출가능 : BOOL; (* AT %MW93011.9 *)
    BB_MAIN_O_통신_CHK : BOOL; (* AT %MW93011.15 *)
    BB_MAIN_O_행거클램프_요구 : BOOL; (* AT %MW93011.8 *)
END_VAR
VAR_EXTERNAL RETAIN
    CLOCK_BIT_1_0Sec : BOOL; (* AT %MW0.5 *) (* CLOCK_BIT_1_0Sec *)
    S369_M_R308_3_언로딩가능 : BOOL; (* AT %MW5004.9 *)
    S369_M_R308_3_클램프완료 : BOOL; (* AT %MW5001.4 *)
    S369_M_R308_3_클램프요구 : BOOL; (* AT %MW5004.11 *)
    S369_M_R308_3_행거안착가능 : BOOL; (* AT %MW5004.10 *)
    S369_M_R308_3_행거안착완료 : BOOL; (* AT %MW5001.3 *)
    S369_M_로딩_이젝터_제품감지_유 : BOOL; (* AT %MW5001.8 *)
    S369_M_언로딩_작업_완료 : BOOL; (* AT %MW5001.1 *)
    S369_M_언로딩버퍼_SEQ : WORD; (* AT %MW10340 *) (* S369 M 언로딩버퍼 SEQ *)
    S369_M_언로딩버퍼_차종_유 : BOOL; (* AT %MW5002.2 *)
    S369_M_운전준비_ON : BOOL; (* AT %MW5000.0 *) (* S369 운전준비 ON *)
    S369_M_자동_운전중 : BOOL; (* AT %MW5000.4 *) (* S369 자동운전중 *)
    S369_M_총괄_SAFETY_이상 : BOOL; (* AT %MW5009.2 *) (* S369_M_총괄_SAFETY_이상 *)
    S369_M_총괄_비상정지_이상 : BOOL; (* AT %MW5009.1 *) (* S369_M_총괄_비상정지_이상 *)
    S369_M_총괄_이상 : BOOL; (* AT %MW5009.0 *) (* S369_M_총괄_이상 *)
END_VAR
VAR
    _e1 : R_TRIG;
END_VAR

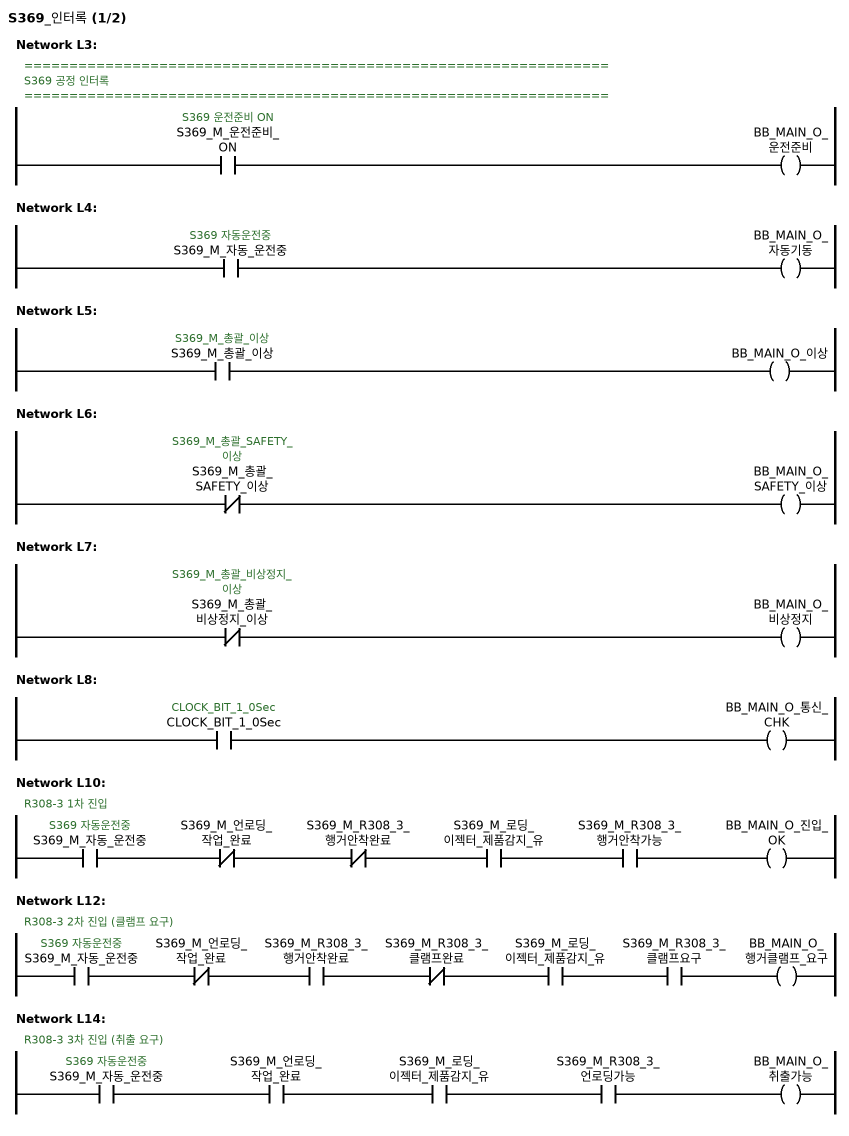
(* ================================================================= *)
(* S369 공정 인터록 *)
(* ================================================================= *)
(* Rung L3 *)
BB_MAIN_O_운전준비 := S369_M_운전준비_ON;
(* Rung L4 *)
BB_MAIN_O_자동기동 := S369_M_자동_운전중;
(* Rung L5 *)
BB_MAIN_O_이상 := S369_M_총괄_이상;
(* Rung L6 *)
BB_MAIN_O_SAFETY_이상 := NOT S369_M_총괄_SAFETY_이상;
(* Rung L7 *)
BB_MAIN_O_비상정지 := NOT S369_M_총괄_비상정지_이상;
(* Rung L8 *)
BB_MAIN_O_통신_CHK := CLOCK_BIT_1_0Sec;
(* R308-3 1차 진입 *)
(* Rung L10 *)
BB_MAIN_O_진입_OK := S369_M_자동_운전중 AND NOT S369_M_언로딩_작업_완료 AND NOT S369_M_R308_3_행거안착완료 AND S369_M_로딩_이젝터_제품감지_유 AND S369_M_R308_3_행거안착가능;
(* R308-3 2차 진입 (클램프 요구) *)
(* Rung L12 *)
BB_MAIN_O_행거클램프_요구 := S369_M_자동_운전중 AND NOT S369_M_언로딩_작업_완료 AND S369_M_R308_3_행거안착완료 AND NOT S369_M_R308_3_클램프완료 AND S369_M_로딩_이젝터_제품감지_유 AND S369_M_R308_3_클램프요구;
(* R308-3 3차 진입 (취출 요구) *)
(* Rung L14 *)
BB_MAIN_O_취출가능 := S369_M_자동_운전중 AND S369_M_언로딩_작업_완료 AND S369_M_로딩_이젝터_제품감지_유 AND S369_M_R308_3_언로딩가능;

